LIN {X 0,Y 340.496,Z 607.338,A -85,B 0,C 180,E1 -14141.61,E2 -14141.61} C_VEL
LIN {X 0,Y 341.817,Z 599.412,A -85,B 0,C 180,E1 -14143.677,E2 -14143.677} C_VEL
LIN {X 0,Y 343.018,Z 591.082,A -85,B 0,C 180,E1 -14145.447,E2 -14145.447} C_VEL
LIN {X 0,Y 344.894,Z 580.855,A -85,B 0,C 180,E1 -14147.186,E2 -14147.186} C_VEL
LIN {X 0,Y 346.926,Z 569.542,A -85,B 0,C 180,E1 -14148.759,E2 -14148.759} C_VEL
LIN {X 0,Y 348.186,Z 560.989,A -85,B 0,C 180,E1 -14149.761,E2 -14149.761} C_VEL
LIN {X 0,Y 348.394,Z 548.85,A -85,B 0,C 180,E1 -14151.085,E2 -14151.085} C_VEL
LIN {X 0,Y 347.208,Z 537.307,A -85,B 0,C 180,E1 -14152.297,E2 -14152.297} C_VEL
LIN {X 0,Y 344.797,Z 525.984,A -85,B 0,C 180,E1 -14153.475,E2 -14153.475} C_VEL
LIN {X 0,Y 341.926,Z 516.235,A -85,B 0,C 180,E1 -14154.518,E2 -14154.518} C_VEL
LIN {X 0,Y 340.89,Z 512.472,A -85,B 0,C 180,E1 -14154.888,E2 -14154.888} C_VEL
LIN {X 0,Y 341.816,Z 505.786,A -85,B 0,C 180,E1 -14158.893,E2 -14158.893} C_VEL
LIN {X 0,Y 342.723,Z 500.774,A -85,B 0,C 180,E1 -14162.22,E2 -14162.22} C_VEL
LIN {X 0,Y 343.565,Z 496.904,A -85,B 0,C 180,E1 -14165.09,E2 -14165.09} C_VEL
LIN {X 0,Y 343.924,Z 493.78,A -85,B 0,C 180,E1 -14167.81,E2 -14167.81} C_VEL
LIN {X 0,Y 343.664,Z 490.982,A -85,B 0,C 180,E1 -14170.875,E2 -14170.875} C_VEL
LIN {X 0,Y 343.334,Z 488.645,A -85,B 0,C 180,E1 -14174.238,E2 -14174.238} C_VEL
LIN {X 0,Y 343.008,Z 487.085,A -85,B 0,C 180,E1 -14177.529,E2 -14177.529} C_VEL
LIN {X 0,Y 342.738,Z 486.117,A -85,B 0,C 180,E1 -14181.188,E2 -14181.188} C_VEL
LIN {X 0,Y 342.591,Z 485.893,A -85,B 0,C 180,E1 -14183.494,E2 -14183.494} C_VEL
LIN {X 0,Y 342.084,Z 486.185,A -85,B 0,C 180,E1 -14187.387,E2 -14187.387} C_VEL
LIN {X 0,Y 341.651,Z 486.869,A -85,B 0,C 180,E1 -14190.416,E2 -14190.416} C_VEL
LIN {X 0,Y 341.105,Z 488.27,A -85,B 0,C 180,E1 -14194.363,E2 -14194.363} C_VEL
LIN {X 0,Y 341.043,Z 488.663,A -85,B 0,C 180,E1 -14195.293,E2 -14195.293} C_VEL
LIN {X 0,Y 341.67,Z 490.745,A -85,B 0,C 180,E1 -14195.532,E2 -14195.532} C_VEL
LIN {X 0,Y 344.946,Z 496.905,A -85,B 0,C 180,E1 -14196.469,E2 -14196.469} C_VEL
LIN {X 0,Y 349.037,Z 506.791,A -85,B 0,C 180,E1 -14197.855,E2 -14197.855} C_VEL
LIN {X 0,Y 351.652,Z 516.211,A -85,B 0,C 180,E1 -14199.095,E2 -14199.095} C_VEL
LIN {X 0,Y 352.15,Z 518.968,A -85,B 0,C 180,E1 -14199.449,E2 -14199.449} C_VEL
LIN {X 0,Y 350.175,Z 531.633,A -85,B 0,C 180,E1 -14200.78,E2 -14200.78} C_VEL
LIN {X 0,Y 348.44,Z 541.84,A -85,B 0,C 180,E1 -14202.119,E2 -14202.119} C_VEL
LIN {X 0,Y 346.392,Z 552.222,A -85,B 0,C 180,E1 -14203.801,E2 -14203.801} C_VEL
LIN {X 0,Y 344.984,Z 559.521,A -85,B 0,C 180,E1 -14205.247,E2 -14205.247} C_VEL
LIN {X 0,Y 343.488,Z 566.818,A -85,B 0,C 180,E1 -14206.993,E2 -14206.993} C_VEL
LIN {X 0,Y 342.385,Z 572.658,A -85,B 0,C 180,E1 -14208.755,E2 -14208.755} C_VEL
LIN {X 0,Y 341.397,Z 577.333,A -85,B 0,C 180,E1 -14210.521,E2 -14210.521} C_VEL
LIN {X 0,Y 340.811,Z 580.1,A -85,B 0,C 180,E1 -14211.823,E2 -14211.823} C_VEL
LIN {X 0,Y 340.324,Z 581.969,A -85,B 0,C 180,E1 -14212.883,E2 -14212.883} C_VEL
LIN {X 0,Y 340.031,Z 583.601,A -85,B 0,C 180,E1 -14214.069,E2 -14214.069} C_VEL
LIN {X 0,Y 339.966,Z 584.783,A -85,B 0,C 180,E1 -14215.257,E2 -14215.257} C_VEL
LIN {X 0,Y 339.738,Z 585.596,A -85,B 0,C 180,E1 -14216.442,E2 -14216.442} C_VEL
LIN {X 0,Y 339.542,Z 586.02,A -85,B 0,C 180,E1 -14217.628,E2 -14217.628} C_VEL
LIN {X 0,Y 339.404,Z 586.008,A -85,B 0,C 180,E1 -14218.814,E2 -14218.814} C_VEL
LIN {X 0,Y 339.34,Z 585.584,A -85,B 0,C 180,E1 -14220,E2 -14220} C_VEL
LIN {X 0,Y 339.328,Z 584.764,A -85,B 0,C 180,E1 -14221.187,E2 -14221.187} C_VEL
LIN {X 0,Y 339.33,Z 583.537,A -85,B 0,C 180,E1 -14222.374,E2 -14222.374} C_VEL
LIN {X 0,Y 339.395,Z 580.863,A -85,B 0,C 180,E1 -14224.157,E2 -14224.157} C_VEL
LIN {X 0,Y 339.641,Z 576.209,A -85,B 0,C 180,E1 -14226.32,E2 -14226.32} C_VEL
LIN {X 0,Y 340.017,Z 570.447,A -85,B 0,C 180,E1 -14228.319,E2 -14228.319} C_VEL
LIN {X 0,Y 340.568,Z 563.931,A -85,B 0,C 180,E1 -14230.103,E2 -14230.103} C_VEL
LIN {X 0,Y 341.218,Z 555.819,A -85,B 0,C 180,E1 -14231.887,E2 -14231.887} C_VEL
LIN {X 0,Y 342.13,Z 545.839,A -85,B 0,C 180,E1 -14233.665,E2 -14233.665} C_VEL
LIN {X 0,Y 343.114,Z 535.532,A -85,B 0,C 180,E1 -14235.139,E2 -14235.139} C_VEL
LIN {X 0,Y 343.987,Z 523.853,A -85,B 0,C 180,E1 -14236.498,E2 -14236.498} C_VEL
LIN {X 0,Y 344.746,Z 513.136,A -85,B 0,C 180,E1 -14237.5,E2 -14237.5} C_VEL
LIN {X 0,Y 345.031,Z 508.34,A -85,B 0,C 180,E1 -14237.884,E2 -14237.884} C_VEL
LIN {X 0,Y 342.241,Z 494.577,A -85,B 0,C 180,E1 -14238.919,E2 -14238.919} C_VEL
LIN {X 0,Y 339.504,Z 481.107,A -85,B 0,C 180,E1 -14239.697,E2 -14239.697} C_VEL
LIN {X 0,Y 339.529,Z 477.775,A -85,B 0,C 180,E1 -14243.16,E2 -14243.16} C_VEL
LIN {X 0,Y 339.735,Z 474.171,A -85,B 0,C 180,E1 -14247.072,E2 -14247.072} C_VEL
LIN {X 0,Y 340.04,Z 474.128,A -85,B 0,C 180,E1 -14249.765,E2 -14249.765} C_VEL
LIN {X 0,Y 340.297,Z 474.098,A -85,B 0,C 180,E1 -14252.478,E2 -14252.478} C_VEL
LIN {X 0,Y 340.557,Z 474.061,A -85,B 0,C 180,E1 -14255.299,E2 -14255.299} C_VEL
LIN {X 0,Y 340.706,Z 474.047,A -85,B 0,C 180,E1 -14258.385,E2 -14258.385} C_VEL
LIN {X 0,Y 340.703,Z 474.046,A -85,B 0,C 180,E1 -14262.046,E2 -14262.046} C_VEL
LIN {X 0,Y 340.656,Z 474.054,A -85,B 0,C 180,E1 -14266.227,E2 -14266.227} C_VEL
LIN {X 0,Y 340.692,Z 474.046,A -85,B 0,C 180,E1 -14269.753,E2 -14269.753} C_VEL
LIN {X 0,Y 340.711,Z 474.041,A -85,B 0,C 180,E1 -14273.259,E2 -14273.259} C_VEL
LIN {X 0,Y 340.698,Z 474.049,A -85,B 0,C 180,E1 -14276.154,E2 -14276.154} C_VEL
LIN {X 0,Y 340.779,Z 474.038,A -85,B 0,C 180,E1 -14280.333,E2 -14280.333} C_VEL
LIN {X 0,Y 340.809,Z 474.03,A -85,B 0,C 180,E1 -14283.02,E2 -14283.02} C_VEL
LIN {X 0,Y 340.733,Z 474.039,A -85,B 0,C 180,E1 -14286.927,E2 -14286.927} C_VEL
LIN {X 0,Y 340.799,Z 474.032,A -85,B 0,C 180,E1 -14290.734,E2 -14290.734} C_VEL
LIN {X 0,Y 340.791,Z 474.032,A -85,B 0,C 180,E1 -14293.219,E2 -14293.219} C_VEL
LIN {X 0,Y 340.849,Z 474.025,A -85,B 0,C 180,E1 -14296.891,E2 -14296.891} C_VEL
LIN {X 0,Y 340.933,Z 474.016,A -85,B 0,C 180,E1 -14300.508,E2 -14300.508} C_VEL
LIN {X 0,Y 341.081,Z 473.996,A -85,B 0,C 180,E1 -14302.898,E2 -14302.898} C_VEL
LIN {X 0,Y 341.173,Z 473.987,A -85,B 0,C 180,E1 -14307.639,E2 -14307.639} C_VEL
LIN {X 0,Y 341.3,Z 473.974,A -85,B 0,C 180,E1 -14310,E2 -14310} C_VEL
LIN {X 0,Y 341.173,Z 473.986,A -85,B 0,C 180,E1 -14312.361,E2 -14312.361} C_VEL
LIN {X 0,Y 341.021,Z 474.003,A -85,B 0,C 180,E1 -14317.103,E2 -14317.103} C_VEL
LIN {X 0,Y 340.875,Z 474.022,A -85,B 0,C 180,E1 -14320.694,E2 -14320.694} C_VEL
LIN {X 0,Y 340.868,Z 474.024,A -85,B 0,C 180,E1 -14324.325,E2 -14324.325} C_VEL
LIN {X 0,Y 340.843,Z 474.027,A -85,B 0,C 180,E1 -14328.467,E2 -14328.467} C_VEL
LIN {X 0,Y 340.726,Z 474.045,A -85,B 0,C 180,E1 -14331.843,E2 -14331.843} C_VEL
LIN {X 0,Y 340.776,Z 474.038,A -85,B 0,C 180,E1 -14335.664,E2 -14335.664} C_VEL
LIN {X 0,Y 340.732,Z 474.041,A -85,B 0,C 180,E1 -14338.321,E2 -14338.321} C_VEL
LIN {X 0,Y 340.702,Z 474.043,A -85,B 0,C 180,E1 -14341.044,E2 -14341.044} C_VEL
LIN {X 0,Y 340.723,Z 474.042,A -85,B 0,C 180,E1 -14345.278,E2 -14345.278} C_VEL
LIN {X 0,Y 340.716,Z 474.042,A -85,B 0,C 180,E1 -14348.386,E2 -14348.386} C_VEL
LIN {X 0,Y 340.703,Z 474.046,A -85,B 0,C 180,E1 -14352.045,E2 -14352.045} C_VEL
LIN {X 0,Y 340.656,Z 474.05,A -85,B 0,C 180,E1 -14356.227,E2 -14356.227} C_VEL
LIN {X 0,Y 340.693,Z 474.05,A -85,B 0,C 180,E1 -14359.752,E2 -14359.752} C_VEL
LIN {X 0,Y 340.687,Z 474.046,A -85,B 0,C 180,E1 -14363.256,E2 -14363.256} C_VEL
LIN {X 0,Y 340.533,Z 474.066,A -85,B 0,C 180,E1 -14366.135,E2 -14366.135} C_VEL
LIN {X 0,Y 340.22,Z 474.103,A -85,B 0,C 180,E1 -14368.906,E2 -14368.906} C_VEL
LIN {X 0,Y 339.997,Z 474.131,A -85,B 0,C 180,E1 -14370.677,E2 -14370.677} C_VEL
LIN {X 0,Y 339.191,Z 474.237,A -85,B 0,C 180,E1 -14371.664,E2 -14371.664} C_VEL
LIN {X 0,Y 336.119,Z 474.617,A -85,B 0,C 180,E1 -14373.265,E2 -14373.265} C_VEL
LIN {X 0,Y 333.569,Z 475.163,A -85,B 0,C 180,E1 -14374.556,E2 -14374.556} C_VEL
LIN {X 0,Y 332.468,Z 475.886,A -85,B 0,C 180,E1 -14375.552,E2 -14375.552} C_VEL
LIN {X 0,Y 332.372,Z 476.217,A -85,B 0,C 180,E1 -14375.888,E2 -14375.888} C_VEL
LIN {X 0,Y 332.378,Z 480.517,A -85,B 0,C 180,E1 -14379.903,E2 -14379.903} C_VEL
LIN {X 0,Y 332.379,Z 480.826,A -85,B 0,C 180,E1 -14380.185,E2 -14380.185} C_VEL
LIN {X 0,Y 335.524,Z 496.725,A -85,B 0,C 180,E1 -14381.146,E2 -14381.146} C_VEL
LIN {X 0,Y 337.973,Z 509.393,A -85,B 0,C 180,E1 -14382.138,E2 -14382.138} C_VEL
LIN {X 0,Y 337.084,Z 521.968,A -85,B 0,C 180,E1 -14383.274,E2 -14383.274} C_VEL
LIN {X 0,Y 336.139,Z 534.349,A -85,B 0,C 180,E1 -14384.694,E2 -14384.694} C_VEL
LIN {X 0,Y 335.24,Z 543.893,A -85,B 0,C 180,E1 -14386.049,E2 -14386.049} C_VEL
LIN {X 0,Y 334.219,Z 554.344,A -85,B 0,C 180,E1 -14387.861,E2 -14387.861} C_VEL
LIN {X 0,Y 333.528,Z 562.727,A -85,B 0,C 180,E1 -14389.682,E2 -14389.682} C_VEL
LIN {X 0,Y 332.939,Z 569.529,A -85,B 0,C 180,E1 -14391.502,E2 -14391.502} C_VEL
LIN {X 0,Y 332.624,Z 574.779,A -85,B 0,C 180,E1 -14393.249,E2 -14393.249} C_VEL
LIN {X 0,Y 332.393,Z 579.258,A -85,B 0,C 180,E1 -14395.148,E2 -14395.148} C_VEL
LIN {X 0,Y 332.264,Z 581.475,A -85,B 0,C 180,E1 -14396.362,E2 -14396.362} C_VEL
LIN {X 0,Y 332.225,Z 583.247,A -85,B 0,C 180,E1 -14397.575,E2 -14397.575} C_VEL
LIN {X 0,Y 332.196,Z 584.613,A -85,B 0,C 180,E1 -14398.787,E2 -14398.787} C_VEL
LIN {X 0,Y 332.235,Z 585.528,A -85,B 0,C 180,E1 -14400,E2 -14400} C_VEL
LIN {X 0,Y 332.48,Z 586.136,A -85,B 0,C 180,E1 -14402.423,E2 -14402.423} C_VEL
LIN {X 0,Y 332.69,Z 585.836,A -85,B 0,C 180,E1 -14403.633,E2 -14403.633} C_VEL
LIN {X 0,Y 332.841,Z 585.101,A -85,B 0,C 180,E1 -14404.845,E2 -14404.845} C_VEL
LIN {X 0,Y 332.912,Z 583.989,A -85,B 0,C 180,E1 -14406.059,E2 -14406.059} C_VEL
LIN {X 0,Y 333.748,Z 580.936,A -85,B 0,C 180,E1 -14408.222,E2 -14408.222} C_VEL
LIN {X 0,Y 334.66,Z 576.679,A -85,B 0,C 180,E1 -14410.282,E2 -14410.282} C_VEL
LIN {X 0,Y 335.8,Z 571.755,A -85,B 0,C 180,E1 -14412.081,E2 -14412.081} C_VEL
LIN {X 0,Y 337.049,Z 565.63,A -85,B 0,C 180,E1 -14413.874,E2 -14413.874} C_VEL
LIN {X 0,Y 338.647,Z 558.164,A -85,B 0,C 180,E1 -14415.652,E2 -14415.652} C_VEL
LIN {X 0,Y 340.629,Z 548.877,A -85,B 0,C 180,E1 -14417.408,E2 -14417.408} C_VEL
LIN {X 0,Y 342.603,Z 538.877,A -85,B 0,C 180,E1 -14418.944,E2 -14418.944} C_VEL
LIN {X 0,Y 344.492,Z 528.159,A -85,B 0,C 180,E1 -14420.293,E2 -14420.293} C_VEL
LIN {X 0,Y 345.869,Z 519.994,A -85,B 0,C 180,E1 -14421.142,E2 -14421.142} C_VEL
LIN {X 0,Y 344.09,Z 511.553,A -85,B 0,C 180,E1 -14422.28,E2 -14422.28} C_VEL
LIN {X 0,Y 340.643,Z 501.465,A -85,B 0,C 180,E1 -14423.708,E2 -14423.708} C_VEL
LIN {X 0,Y 335.961,Z 491.247,A -85,B 0,C 180,E1 -14425.26,E2 -14425.26} C_VEL
LIN {X 0,Y 334.34,Z 488.16,A -85,B 0,C 180,E1 -14425.755,E2 -14425.755} C_VEL
LIN {X 0,Y 334.158,Z 487.37,A -85,B 0,C 180,E1 -14425.866,E2 -14425.866} C_VEL
LIN {X 0,Y 334.333,Z 484.941,A -85,B 0,C 180,E1 -14428.913,E2 -14428.913} C_VEL
LIN {X 0,Y 334.598,Z 482.863,A -85,B 0,C 180,E1 -14431.675,E2 -14431.675} C_VEL
LIN {X 0,Y 334.724,Z 480.616,A -85,B 0,C 180,E1 -14435.029,E2 -14435.029} C_VEL
LIN {X 0,Y 334.588,Z 479.264,A -85,B 0,C 180,E1 -14437.528,E2 -14437.528} C_VEL
LIN {X 0,Y 334.37,Z 477.929,A -85,B 0,C 180,E1 -14440.828,E2 -14440.828} C_VEL
LIN {X 0,Y 334.191,Z 477.226,A -85,B 0,C 180,E1 -14444.355,E2 -14444.355} C_VEL
LIN {X 0,Y 334.119,Z 477.409,A -85,B 0,C 180,E1 -14446.387,E2 -14446.387} C_VEL
LIN {X 0,Y 335.222,Z 483.366,A -85,B 0,C 180,E1 -14450.197,E2 -14450.197} C_VEL
LIN {X 0,Y 335.855,Z 487.414,A -85,B 0,C 180,E1 -14452.672,E2 -14452.672} C_VEL
LIN {X 0,Y 335.789,Z 490.904,A -85,B 0,C 180,E1 -14454.712,E2 -14454.712} C_VEL
LIN {X 0,Y 334.967,Z 497.396,A -85,B 0,C 180,E1 -14458.363,E2 -14458.363} C_VEL
LIN {X 0,Y 334.076,Z 504.808,A -85,B 0,C 180,E1 -14462.431,E2 -14462.431} C_VEL
LIN {X 0,Y 333.699,Z 508.242,A -85,B 0,C 180,E1 -14464.212,E2 -14464.212} C_VEL
LIN {X 0,Y 334.485,Z 512.006,A -85,B 0,C 180,E1 -14464.578,E2 -14464.578} C_VEL
LIN {X 0,Y 335.342,Z 514.335,A -85,B 0,C 180,E1 -14464.855,E2 -14464.855} C_VEL
LIN {X 0,Y 338.443,Z 526.565,A -85,B 0,C 180,E1 -14466.171,E2 -14466.171} C_VEL
LIN {X 0,Y 340.605,Z 539.432,A -85,B 0,C 180,E1 -14467.544,E2 -14467.544} C_VEL
LIN {X 0,Y 341.392,Z 550.711,A -85,B 0,C 180,E1 -14468.783,E2 -14468.783} C_VEL
LIN {X 0,Y 341.006,Z 563.3,A -85,B 0,C 180,E1 -14470.276,E2 -14470.276} C_VEL
LIN {X 0,Y 339.006,Z 574.502,A -85,B 0,C 180,E1 -14471.726,E2 -14471.726} C_VEL
LIN {X 0,Y 337.173,Z 584.837,A -85,B 0,C 180,E1 -14473.374,E2 -14473.374} C_VEL
LIN {X 0,Y 335.767,Z 592.423,A -85,B 0,C 180,E1 -14474.833,E2 -14474.833} C_VEL
LIN {X 0,Y 334.486,Z 600.221,A -85,B 0,C 180,E1 -14476.637,E2 -14476.637} C_VEL
LIN {X 0,Y 333.373,Z 606.607,A -85,B 0,C 180,E1 -14478.447,E2 -14478.447} C_VEL
LIN {X 0,Y 332.716,Z 611.78,A -85,B 0,C 180,E1 -14480.271,E2 -14480.271} C_VEL
LIN {X 0,Y 332.326,Z 615.858,A -85,B 0,C 180,E1 -14482.099,E2 -14482.099} C_VEL
LIN {X 0,Y 332.18,Z 618.907,A -85,B 0,C 180,E1 -14483.928,E2 -14483.928} C_VEL
LIN {X 0,Y 332.114,Z 620.392,A -85,B 0,C 180,E1 -14485.144,E2 -14485.144} C_VEL
LIN {X 0,Y 332.104,Z 621.472,A -85,B 0,C 180,E1 -14486.36,E2 -14486.36} C_VEL
LIN {X 0,Y 332.293,Z 623.081,A -85,B 0,C 180,E1 -14488.788,E2 -14488.788} C_VEL
LIN {X 0,Y 332.277,Z 623.714,A -85,B 0,C 180,E1 -14490,E2 -14490} C_VEL
LIN {X 0,Y 332.252,Z 623.93,A -85,B 0,C 180,E1 -14491.212,E2 -14491.212} C_VEL
LIN {X 0,Y 332.081,Z 623.725,A -85,B 0,C 180,E1 -14492.426,E2 -14492.426} C_VEL
LIN {X 0,Y 332.058,Z 623.108,A -85,B 0,C 180,E1 -14493.64,E2 -14493.64} C_VEL
LIN {X 0,Y 332.045,Z 620.869,A -85,B 0,C 180,E1 -14495.848,E2 -14495.848} C_VEL
LIN {X 0,Y 332.321,Z 617.551,A -85,B 0,C 180,E1 -14497.901,E2 -14497.901} C_VEL
LIN {X 0,Y 332.748,Z 613.523,A -85,B 0,C 180,E1 -14499.728,E2 -14499.728} C_VEL
LIN {X 0,Y 333.403,Z 608.444,A -85,B 0,C 180,E1 -14501.552,E2 -14501.552} C_VEL
LIN {X 0,Y 334.727,Z 601.005,A -85,B 0,C 180,E1 -14503.663,E2 -14503.663} C_VEL
LIN {X 0,Y 335.98,Z 593.086,A -85,B 0,C 180,E1 -14505.468,E2 -14505.468} C_VEL
LIN {X 0,Y 337.879,Z 583.553,A -85,B 0,C 180,E1 -14507.242,E2 -14507.242} C_VEL
LIN {X 0,Y 339.924,Z 572.979,A -85,B 0,C 180,E1 -14508.848,E2 -14508.848} C_VEL
LIN {X 0,Y 341.693,Z 562.538,A -85,B 0,C 180,E1 -14510.152,E2 -14510.152} C_VEL
LIN {X 0,Y 342.125,Z 551.121,A -85,B 0,C 180,E1 -14511.491,E2 -14511.491} C_VEL
LIN {X 0,Y 341.157,Z 539.755,A -85,B 0,C 180,E1 -14512.757,E2 -14512.757} C_VEL
LIN {X 0,Y 339.073,Z 528.891,A -85,B 0,C 180,E1 -14513.987,E2 -14513.987} C_VEL
LIN {X 0,Y 335.758,Z 516.942,A -85,B 0,C 180,E1 -14515.361,E2 -14515.361} C_VEL
LIN {X 0,Y 334.191,Z 512.494,A -85,B 0,C 180,E1 -14515.897,E2 -14515.897} C_VEL
LIN {X 0,Y 334.081,Z 511.612,A -85,B 0,C 180,E1 -14516.01,E2 -14516.01} C_VEL
LIN {X 0,Y 334.958,Z 505.999,A -85,B 0,C 180,E1 -14519.543,E2 -14519.543} C_VEL
LIN {X 0,Y 336.044,Z 500.735,A -85,B 0,C 180,E1 -14523.222,E2 -14523.222} C_VEL
LIN {X 0,Y 336.707,Z 497.527,A -85,B 0,C 180,E1 -14525.763,E2 -14525.763} C_VEL
LIN {X 0,Y 336.986,Z 495.505,A -85,B 0,C 180,E1 -14527.579,E2 -14527.579} C_VEL
LIN {X 0,Y 336.771,Z 492.993,A -85,B 0,C 180,E1 -14530.311,E2 -14530.311} C_VEL
LIN {X 0,Y 336.456,Z 490.624,A -85,B 0,C 180,E1 -14533.576,E2 -14533.576} C_VEL
LIN {X 0,Y 336.131,Z 488.849,A -85,B 0,C 180,E1 -14537.038,E2 -14537.038} C_VEL
LIN {X 0,Y 335.843,Z 487.754,A -85,B 0,C 180,E1 -14540.74,E2 -14540.74} C_VEL
LIN {X 0,Y 335.563,Z 487.416,A -85,B 0,C 180,E1 -14544.096,E2 -14544.096} C_VEL
LIN {X 0,Y 335.191,Z 487.593,A -85,B 0,C 180,E1 -14547.002,E2 -14547.002} C_VEL
LIN {X 0,Y 334.819,Z 488.108,A -85,B 0,C 180,E1 -14549.75,E2 -14549.75} C_VEL
LIN {X 0,Y 334.374,Z 488.911,A -85,B 0,C 180,E1 -14552.458,E2 -14552.458} C_VEL
LIN {X 0,Y 334.19,Z 489.753,A -85,B 0,C 180,E1 -14554.235,E2 -14554.235} C_VEL
LIN {X 0,Y 334.84,Z 491.695,A -85,B 0,C 180,E1 -14554.493,E2 -14554.493} C_VEL
LIN {X 0,Y 336.559,Z 494.566,A -85,B 0,C 180,E1 -14555,E2 -14555} C_VEL
LIN {X 0,Y 341.643,Z 505.533,A -85,B 0,C 180,E1 -14556.726,E2 -14556.726} C_VEL
LIN {X 0,Y 344.431,Z 513.763,A -85,B 0,C 180,E1 -14557.939,E2 -14557.939} C_VEL
LIN {X 0,Y 345.962,Z 520.424,A -85,B 0,C 180,E1 -14558.865,E2 -14558.865} C_VEL
LIN {X 0,Y 344.002,Z 532.862,A -85,B 0,C 180,E1 -14560.242,E2 -14560.242} C_VEL
LIN {X 0,Y 341.96,Z 543.699,A -85,B 0,C 180,E1 -14561.735,E2 -14561.735} C_VEL
LIN {X 0,Y 339.778,Z 554.044,A -85,B 0,C 180,E1 -14563.477,E2 -14563.477} C_VEL
LIN {X 0,Y 337.997,Z 562.331,A -85,B 0,C 180,E1 -14565.243,E2 -14565.243} C_VEL
LIN {X 0,Y 336.297,Z 570.142,A -85,B 0,C 180,E1 -14567.325,E2 -14567.325} C_VEL
LIN {X 0,Y 335.006,Z 575.464,A -85,B 0,C 180,E1 -14569.117,E2 -14569.117} C_VEL
LIN {X 0,Y 334.179,Z 579.617,A -85,B 0,C 180,E1 -14570.925,E2 -14570.925} C_VEL
LIN {X 0,Y 333.327,Z 582.773,A -85,B 0,C 180,E1 -14572.732,E2 -14572.732} C_VEL
LIN {X 0,Y 332.997,Z 584.305,A -85,B 0,C 180,E1 -14573.943,E2 -14573.943} C_VEL
LIN {X 0,Y 332.933,Z 585.431,A -85,B 0,C 180,E1 -14575.157,E2 -14575.157} C_VEL
LIN {X 0,Y 332.699,Z 586.188,A -85,B 0,C 180,E1 -14576.367,E2 -14576.367} C_VEL
LIN {X 0,Y 332.491,Z 586.523,A -85,B 0,C 180,E1 -14577.577,E2 -14577.577} C_VEL
LIN {X 0,Y 332.346,Z 586.435,A -85,B 0,C 180,E1 -14578.789,E2 -14578.789} C_VEL
LIN {X 0,Y 332.261,Z 585.954,A -85,B 0,C 180,E1 -14580,E2 -14580} C_VEL
LIN {X 0,Y 332.236,Z 585.078,A -85,B 0,C 180,E1 -14581.212,E2 -14581.212} C_VEL
LIN {X 0,Y 332.235,Z 583.755,A -85,B 0,C 180,E1 -14582.425,E2 -14582.425} C_VEL
LIN {X 0,Y 332.329,Z 580.982,A -85,B 0,C 180,E1 -14584.245,E2 -14584.245} C_VEL
LIN {X 0,Y 332.528,Z 577.163,A -85,B 0,C 180,E1 -14586.066,E2 -14586.066} C_VEL
LIN {X 0,Y 332.844,Z 572.204,A -85,B 0,C 180,E1 -14587.889,E2 -14587.889} C_VEL
LIN {X 0,Y 333.429,Z 564.814,A -85,B 0,C 180,E1 -14590.015,E2 -14590.015} C_VEL
LIN {X 0,Y 334.106,Z 556.824,A -85,B 0,C 180,E1 -14591.835,E2 -14591.835} C_VEL
LIN {X 0,Y 335.012,Z 546.946,A -85,B 0,C 180,E1 -14593.651,E2 -14593.651} C_VEL
LIN {X 0,Y 335.997,Z 536.831,A -85,B 0,C 180,E1 -14595.157,E2 -14595.157} C_VEL
LIN {X 0,Y 336.898,Z 525.046,A -85,B 0,C 180,E1 -14596.579,E2 -14596.579} C_VEL
LIN {X 0,Y 337.777,Z 513.253,A -85,B 0,C 180,E1 -14597.716,E2 -14597.716} C_VEL
LIN {X 0,Y 337.941,Z 508.65,A -85,B 0,C 180,E1 -14598.099,E2 -14598.099} C_VEL
LIN {X 0,Y 335.191,Z 495.352,A -85,B 0,C 180,E1 -14599.12,E2 -14599.12} C_VEL
LIN {X 0,Y 332.429,Z 481.496,A -85,B 0,C 180,E1 -14599.932,E2 -14599.932} C_VEL
LIN {X 0,Y 332.467,Z 477.936,A -85,B 0,C 180,E1 -14603.681,E2 -14603.681} C_VEL
LIN {X 0,Y 332.597,Z 475.452,A -85,B 0,C 180,E1 -14606.344,E2 -14606.344} C_VEL
LIN {X 0,Y 332.736,Z 475.044,A -85,B 0,C 180,E1 -14607.69,E2 -14607.69} C_VEL
LIN {X 0,Y 333.033,Z 475.003,A -85,B 0,C 180,E1 -14610.43,E2 -14610.43} C_VEL
LIN {X 0,Y 333.306,Z 474.964,A -85,B 0,C 180,E1 -14613.246,E2 -14613.246} C_VEL
LIN {X 0,Y 333.635,Z 474.924,A -85,B 0,C 180,E1 -14616.825,E2 -14616.825} C_VEL
LIN {X 0,Y 333.651,Z 474.923,A -85,B 0,C 180,E1 -14620.685,E2 -14620.685} C_VEL
LIN {X 0,Y 333.598,Z 474.933,A -85,B 0,C 180,E1 -14624.251,E2 -14624.251} C_VEL
LIN {X 0,Y 333.645,Z 474.923,A -85,B 0,C 180,E1 -14627.619,E2 -14627.619} C_VEL
LIN {X 0,Y 333.658,Z 474.92,A -85,B 0,C 180,E1 -14631.202,E2 -14631.202} C_VEL
LIN {X 0,Y 333.681,Z 474.92,A -85,B 0,C 180,E1 -14633.861,E2 -14633.861} C_VEL
LIN {X 0,Y 333.65,Z 474.921,A -85,B 0,C 180,E1 -14637.413,E2 -14637.413} C_VEL
LIN {X 0,Y 333.715,Z 474.913,A -85,B 0,C 180,E1 -14641.028,E2 -14641.028} C_VEL
LIN {X 0,Y 333.74,Z 474.912,A -85,B 0,C 180,E1 -14643.754,E2 -14643.754} C_VEL
LIN {X 0,Y 333.724,Z 474.916,A -85,B 0,C 180,E1 -14647.914,E2 -14647.914} C_VEL
LIN {X 0,Y 333.799,Z 474.904,A -85,B 0,C 180,E1 -14651.59,E2 -14651.59} C_VEL
LIN {X 0,Y 333.813,Z 474.902,A -85,B 0,C 180,E1 -14655.577,E2 -14655.577} C_VEL
LIN {X 0,Y 333.839,Z 474.897,A -85,B 0,C 180,E1 -14659.078,E2 -14659.078} C_VEL
LIN {X 0,Y 334.031,Z 474.874,A -85,B 0,C 180,E1 -14662.748,E2 -14662.748} C_VEL
LIN {X 0,Y 333.815,Z 474.901,A -85,B 0,C 180,E1 -14665.169,E2 -14665.169} C_VEL
LIN {X 0,Y 334.11,Z 474.866,A -85,B 0,C 180,E1 -14667.589,E2 -14667.589} C_VEL
LIN {X 0,Y 334.251,Z 474.852,A -85,B 0,C 180,E1 -14670,E2 -14670} C_VEL
LIN {X 0,Y 334.11,Z 474.866,A -85,B 0,C 180,E1 -14672.411,E2 -14672.411} C_VEL
LIN {X 0,Y 334.004,Z 474.882,A -85,B 0,C 180,E1 -14676.039,E2 -14676.039} C_VEL
LIN {X 0,Y 333.853,Z 474.899,A -85,B 0,C 180,E1 -14679.695,E2 -14679.695} C_VEL
LIN {X 0,Y 333.802,Z 474.903,A -85,B 0,C 180,E1 -14683.391,E2 -14683.391} C_VEL
LIN {X 0,Y 333.751,Z 474.909,A -85,B 0,C 180,E1 -14687.146,E2 -14687.146} C_VEL
LIN {X 0,Y 333.74,Z 474.914,A -85,B 0,C 180,E1 -14689.69,E2 -14689.69} C_VEL
LIN {X 0,Y 333.676,Z 474.921,A -85,B 0,C 180,E1 -14693.59,E2 -14693.59} C_VEL
LIN {X 0,Y 333.739,Z 474.912,A -85,B 0,C 180,E1 -14696.246,E2 -14696.246} C_VEL
LIN {X 0,Y 333.694,Z 474.916,A -85,B 0,C 180,E1 -14698.974,E2 -14698.974} C_VEL
LIN {X 0,Y 333.65,Z 474.921,A -85,B 0,C 180,E1 -14702.587,E2 -14702.587} C_VEL
LIN {X 0,Y 333.681,Z 474.92,A -85,B 0,C 180,E1 -14706.138,E2 -14706.138} C_VEL
LIN {X 0,Y 333.651,Z 474.922,A -85,B 0,C 180,E1 -14709.192,E2 -14709.192} C_VEL
LIN {X 0,Y 333.636,Z 474.923,A -85,B 0,C 180,E1 -14712.5,E2 -14712.5} C_VEL
LIN {X 0,Y 333.601,Z 474.931,A -85,B 0,C 180,E1 -14715.955,E2 -14715.955} C_VEL
LIN {X 0,Y 333.651,Z 474.923,A -85,B 0,C 180,E1 -14719.315,E2 -14719.315} C_VEL
LIN {X 0,Y 333.65,Z 474.922,A -85,B 0,C 180,E1 -14723.172,E2 -14723.172} C_VEL
LIN {X 0,Y 333.424,Z 474.949,A -85,B 0,C 180,E1 -14726.767,E2 -14726.767} C_VEL
LIN {X 0,Y 332.955,Z 475.008,A -85,B 0,C 180,E1 -14730.656,E2 -14730.656} C_VEL
LIN {X 0,Y 332.487,Z 475.069,A -85,B 0,C 180,E1 -14734.321,E2 -14734.321} C_VEL
LIN {X 0,Y 332.426,Z 475.264,A -85,B 0,C 180,E1 -14734.986,E2 -14734.986} C_VEL
LIN {X 0,Y 332.372,Z 476.217,A -85,B 0,C 180,E1 -14735.888,E2 -14735.888} C_VEL
LIN {X 0,Y 331.679,Z 476.986,A -85,B 0,C 180,E1 -14736.548,E2 -14736.548} C_VEL
LIN {X 0,Y 328.822,Z 478.348,A -85,B 0,C 180,E1 -14737.577,E2 -14737.577} C_VEL
LIN {X 0,Y 325.963,Z 479.714,A -85,B 0,C 180,E1 -14738.623,E2 -14738.623} C_VEL
LIN {X 0,Y 325.292,Z 480.498,A -85,B 0,C 180,E1 -14739.302,E2 -14739.302} C_VEL
LIN {X 0,Y 325.306,Z 481.171,A -85,B 0,C 180,E1 -14739.929,E2 -14739.929} C_VEL
LIN {X 0,Y 328.254,Z 496.354,A -85,B 0,C 180,E1 -14740.862,E2 -14740.862} C_VEL
LIN {X 0,Y 330.77,Z 509.322,A -85,B 0,C 180,E1 -14741.896,E2 -14741.896} C_VEL
LIN {X 0,Y 330.54,Z 516.482,A -85,B 0,C 180,E1 -14742.522,E2 -14742.522} C_VEL
LIN {X 0,Y 329.538,Z 529.554,A -85,B 0,C 180,E1 -14743.904,E2 -14743.904} C_VEL
LIN {X 0,Y 328.582,Z 540.013,A -85,B 0,C 180,E1 -14745.286,E2 -14745.286} C_VEL
LIN {X 0,Y 327.556,Z 550.469,A -85,B 0,C 180,E1 -14746.98,E2 -14746.98} C_VEL
LIN {X 0,Y 326.74,Z 559.698,A -85,B 0,C 180,E1 -14748.838,E2 -14748.838} C_VEL
LIN {X 0,Y 326.088,Z 567.169,A -85,B 0,C 180,E1 -14750.697,E2 -14750.697} C_VEL
LIN {X 0,Y 325.636,Z 573.186,A -85,B 0,C 180,E1 -14752.559,E2 -14752.559} C_VEL
LIN {X 0,Y 325.39,Z 577.947,A -85,B 0,C 180,E1 -14754.422,E2 -14754.422} C_VEL
LIN {X 0,Y 325.19,Z 581.588,A -85,B 0,C 180,E1 -14756.282,E2 -14756.282} C_VEL
LIN {X 0,Y 325.131,Z 583.422,A -85,B 0,C 180,E1 -14757.522,E2 -14757.522} C_VEL
LIN {X 0,Y 325.101,Z 584.85,A -85,B 0,C 180,E1 -14758.761,E2 -14758.761} C_VEL
LIN {X 0,Y 325.144,Z 585.873,A -85,B 0,C 180,E1 -14760,E2 -14760} C_VEL
LIN {X 0,Y 325.238,Z 586.439,A -85,B 0,C 180,E1 -14761.238,E2 -14761.238} C_VEL
LIN {X 0,Y 325.412,Z 586.605,A -85,B 0,C 180,E1 -14762.475,E2 -14762.475} C_VEL
LIN {X 0,Y 325.63,Z 586.378,A -85,B 0,C 180,E1 -14763.712,E2 -14763.712} C_VEL
LIN {X 0,Y 325.793,Z 585.747,A -85,B 0,C 180,E1 -14764.95,E2 -14764.95} C_VEL
LIN {X 0,Y 325.885,Z 584.708,A -85,B 0,C 180,E1 -14766.19,E2 -14766.19} C_VEL
LIN {X 0,Y 326.781,Z 581.813,A -85,B 0,C 180,E1 -14768.383,E2 -14768.383} C_VEL
LIN {X 0,Y 327.748,Z 577.71,A -85,B 0,C 180,E1 -14770.502,E2 -14770.502} C_VEL
LIN {X 0,Y 328.968,Z 572.965,A -85,B 0,C 180,E1 -14772.335,E2 -14772.335} C_VEL
LIN {X 0,Y 330.32,Z 567.053,A -85,B 0,C 180,E1 -14774.163,E2 -14774.163} C_VEL
LIN {X 0,Y 331.997,Z 559.754,A -85,B 0,C 180,E1 -14775.973,E2 -14775.973} C_VEL
LIN {X 0,Y 334.098,Z 550.84,A -85,B 0,C 180,E1 -14777.759,E2 -14777.759} C_VEL
LIN {X 0,Y 336.469,Z 539.837,A -85,B 0,C 180,E1 -14779.524,E2 -14779.524} C_VEL
LIN {X 0,Y 338.565,Z 528.71,A -85,B 0,C 180,E1 -14780.95,E2 -14780.95} C_VEL
LIN {X 0,Y 339.755,Z 521.85,A -85,B 0,C 180,E1 -14781.7,E2 -14781.7} C_VEL
LIN {X 0,Y 338.006,Z 513.498,A -85,B 0,C 180,E1 -14782.916,E2 -14782.916} C_VEL
LIN {X 0,Y 334.622,Z 503.528,A -85,B 0,C 180,E1 -14784.452,E2 -14784.452} C_VEL
LIN {X 0,Y 331.443,Z 496.294,A -85,B 0,C 180,E1 -14785.628,E2 -14785.628} C_VEL
LIN {X 0,Y 329.103,Z 491.959,A -85,B 0,C 180,E1 -14786.418,E2 -14786.418} C_VEL
LIN {X 0,Y 327.493,Z 488.852,A -85,B 0,C 180,E1 -14786.969,E2 -14786.969} C_VEL
LIN {X 0,Y 327.325,Z 488.186,A -85,B 0,C 180,E1 -14787.059,E2 -14787.059} C_VEL
LIN {X 0,Y 327.697,Z 485.292,A -85,B 0,C 180,E1 -14790.979,E2 -14790.979} C_VEL
LIN {X 0,Y 327.89,Z 483.403,A -85,B 0,C 180,E1 -14793.868,E2 -14793.868} C_VEL
LIN {X 0,Y 327.869,Z 481.787,A -85,B 0,C 180,E1 -14796.883,E2 -14796.883} C_VEL
LIN {X 0,Y 327.698,Z 480.572,A -85,B 0,C 180,E1 -14800.046,E2 -14800.046} C_VEL
LIN {X 0,Y 327.575,Z 479.93,A -85,B 0,C 180,E1 -14803.357,E2 -14803.357} C_VEL
LIN {X 0,Y 327.57,Z 479.849,A -85,B 0,C 180,E1 -14805.073,E2 -14805.073} C_VEL
LIN {X 0,Y 327.456,Z 480.329,A -85,B 0,C 180,E1 -14807.585,E2 -14807.585} C_VEL
LIN {X 0,Y 328.261,Z 484.712,A -85,B 0,C 180,E1 -14810.422,E2 -14810.422} C_VEL
LIN {X 0,Y 328.888,Z 489.273,A -85,B 0,C 180,E1 -14813.249,E2 -14813.249} C_VEL
LIN {X 0,Y 328.581,Z 493.046,A -85,B 0,C 180,E1 -14815.472,E2 -14815.472} C_VEL
LIN {X 0,Y 327.677,Z 499.36,A -85,B 0,C 180,E1 -14819.084,E2 -14819.084} C_VEL
LIN {X 0,Y 326.968,Z 505.398,A -85,B 0,C 180,E1 -14822.475,E2 -14822.475} C_VEL
LIN {X 0,Y 326.883,Z 506.414,A -85,B 0,C 180,E1 -14822.922,E2 -14822.922} C_VEL
LIN {X 0,Y 327.604,Z 510.053,A -85,B 0,C 180,E1 -14823.311,E2 -14823.311} C_VEL
LIN {X 0,Y 328.667,Z 512.658,A -85,B 0,C 180,E1 -14823.669,E2 -14823.669} C_VEL
LIN {X 0,Y 332.104,Z 526.167,A -85,B 0,C 180,E1 -14825.25,E2 -14825.25} C_VEL
LIN {X 0,Y 334.288,Z 539.435,A -85,B 0,C 180,E1 -14826.776,E2 -14826.776} C_VEL
LIN {X 0,Y 335.131,Z 550.563,A -85,B 0,C 180,E1 -14828.083,E2 -14828.083} C_VEL
LIN {X 0,Y 334.614,Z 563.818,A -85,B 0,C 180,E1 -14829.723,E2 -14829.723} C_VEL
LIN {X 0,Y 332.566,Z 574.699,A -85,B 0,C 180,E1 -14831.199,E2 -14831.199} C_VEL
LIN {X 0,Y 330.439,Z 585.664,A -85,B 0,C 180,E1 -14833.027,E2 -14833.027} C_VEL
LIN {X 0,Y 328.945,Z 593.029,A -85,B 0,C 180,E1 -14834.51,E2 -14834.51} C_VEL
LIN {X 0,Y 327.355,Z 601.696,A -85,B 0,C 180,E1 -14836.656,E2 -14836.656} C_VEL
LIN {X 0,Y 326.393,Z 606.798,A -85,B 0,C 180,E1 -14838.196,E2 -14838.196} C_VEL
LIN {X 0,Y 325.705,Z 611.826,A -85,B 0,C 180,E1 -14840.06,E2 -14840.06} C_VEL
LIN {X 0,Y 325.255,Z 615.76,A -85,B 0,C 180,E1 -14841.926,E2 -14841.926} C_VEL
LIN {X 0,Y 325.102,Z 618.902,A -85,B 0,C 180,E1 -14843.945,E2 -14843.945} C_VEL
LIN {X 0,Y 325.027,Z 621.129,A -85,B 0,C 180,E1 -14846.281,E2 -14846.281} C_VEL
LIN {X 0,Y 325.234,Z 622.469,A -85,B 0,C 180,E1 -14848.762,E2 -14848.762} C_VEL
LIN {X 0,Y 325.219,Z 623.191,A -85,B 0,C 180,E1 -14850,E2 -14850} C_VEL
LIN {X 0,Y 325.17,Z 623.453,A -85,B 0,C 180,E1 -14851.238,E2 -14851.238} C_VEL
LIN {X 0,Y 324.98,Z 622.741,A -85,B 0,C 180,E1 -14853.72,E2 -14853.72} C_VEL
LIN {X 0,Y 324.962,Z 620.843,A -85,B 0,C 180,E1 -14855.818,E2 -14855.818} C_VEL
LIN {X 0,Y 325.252,Z 617.449,A -85,B 0,C 180,E1 -14858.074,E2 -14858.074} C_VEL
LIN {X 0,Y 325.737,Z 613.566,A -85,B 0,C 180,E1 -14859.939,E2 -14859.939} C_VEL
LIN {X 0,Y 326.42,Z 608.609,A -85,B 0,C 180,E1 -14861.803,E2 -14861.803} C_VEL
LIN {X 0,Y 327.844,Z 601.33,A -85,B 0,C 180,E1 -14863.955,E2 -14863.955} C_VEL
LIN {X 0,Y 329.16,Z 593.754,A -85,B 0,C 180,E1 -14865.788,E2 -14865.788} C_VEL
LIN {X 0,Y 331.169,Z 584.427,A -85,B 0,C 180,E1 -14867.603,E2 -14867.603} C_VEL
LIN {X 0,Y 333.535,Z 573.185,A -85,B 0,C 180,E1 -14869.383,E2 -14869.383} C_VEL
LIN {X 0,Y 335.238,Z 564.28,A -85,B 0,C 180,E1 -14870.558,E2 -14870.558} C_VEL
LIN {X 0,Y 335.872,Z 553.143,A -85,B 0,C 180,E1 -14871.933,E2 -14871.933} C_VEL
LIN {X 0,Y 335.071,Z 541.555,A -85,B 0,C 180,E1 -14873.328,E2 -14873.328} C_VEL
LIN {X 0,Y 332.849,Z 529.578,A -85,B 0,C 180,E1 -14874.779,E2 -14874.779} C_VEL
LIN {X 0,Y 330.498,Z 520.62,A -85,B 0,C 180,E1 -14875.895,E2 -14875.895} C_VEL
LIN {X 0,Y 328.389,Z 514.694,A -85,B 0,C 180,E1 -14876.707,E2 -14876.707} C_VEL
LIN {X 0,Y 327.324,Z 510.93,A -85,B 0,C 180,E1 -14877.168,E2 -14877.168} C_VEL
LIN {X 0,Y 328.422,Z 504.938,A -85,B 0,C 180,E1 -14881.133,E2 -14881.133} C_VEL
LIN {X 0,Y 329.194,Z 501.459,A -85,B 0,C 180,E1 -14883.716,E2 -14883.716} C_VEL
LIN {X 0,Y 329.892,Z 498.013,A -85,B 0,C 180,E1 -14886.621,E2 -14886.621} C_VEL
LIN {X 0,Y 330.01,Z 496.448,A -85,B 0,C 180,E1 -14888.141,E2 -14888.141} C_VEL
LIN {X 0,Y 329.891,Z 494.849,A -85,B 0,C 180,E1 -14889.92,E2 -14889.92} C_VEL
LIN {X 0,Y 329.559,Z 492.228,A -85,B 0,C 180,E1 -14893.526,E2 -14893.526} C_VEL
LIN {X 0,Y 329.221,Z 490.494,A -85,B 0,C 180,E1 -14896.912,E2 -14896.912} C_VEL
LIN {X 0,Y 328.934,Z 489.424,A -85,B 0,C 180,E1 -14900.28,E2 -14900.28} C_VEL
LIN {X 0,Y 328.704,Z 488.991,A -85,B 0,C 180,E1 -14903.226,E2 -14903.226} C_VEL
LIN {X 0,Y 328.307,Z 489.046,A -85,B 0,C 180,E1 -14906.602,E2 -14906.602} C_VEL
LIN {X 0,Y 327.951,Z 489.408,A -85,B 0,C 180,E1 -14909.048,E2 -14909.048} C_VEL
LIN {X 0,Y 327.316,Z 490.486,A -85,B 0,C 180,E1 -14913.005,E2 -14913.005} C_VEL
LIN {X 0,Y 327.849,Z 492.242,A -85,B 0,C 180,E1 -14913.245,E2 -14913.245} C_VEL
LIN {X 0,Y 329.8,Z 495.191,A -85,B 0,C 180,E1 -14913.864,E2 -14913.864} C_VEL
LIN {X 0,Y 334.993,Z 506.268,A -85,B 0,C 180,E1 -14915.786,E2 -14915.786} C_VEL
LIN {X 0,Y 338.441,Z 516.1,A -85,B 0,C 180,E1 -14917.358,E2 -14917.358} C_VEL
LIN {X 0,Y 339.826,Z 522.46,A -85,B 0,C 180,E1 -14918.321,E2 -14918.321} C_VEL
LIN {X 0,Y 338.895,Z 528.831,A -85,B 0,C 180,E1 -14919.04,E2 -14919.04} C_VEL
LIN {X 0,Y 336.696,Z 540.149,A -85,B 0,C 180,E1 -14920.49,E2 -14920.49} C_VEL
LIN {X 0,Y 334.655,Z 549.468,A -85,B 0,C 180,E1 -14921.955,E2 -14921.955} C_VEL
LIN {X 0,Y 332.467,Z 558.693,A -85,B 0,C 180,E1 -14923.735,E2 -14923.735} C_VEL
LIN {X 0,Y 330.452,Z 567.356,A -85,B 0,C 180,E1 -14925.843,E2 -14925.843} C_VEL
LIN {X 0,Y 329.09,Z 573.262,A -85,B 0,C 180,E1 -14927.669,E2 -14927.669} C_VEL
LIN {X 0,Y 327.863,Z 578,A -85,B 0,C 180,E1 -14929.502,E2 -14929.502} C_VEL
LIN {X 0,Y 326.901,Z 581.902,A -85,B 0,C 180,E1 -14931.476,E2 -14931.476} C_VEL
LIN {X 0,Y 326.334,Z 583.585,A -85,B 0,C 180,E1 -14932.576,E2 -14932.576} C_VEL
LIN {X 0,Y 325.97,Z 585.047,A -85,B 0,C 180,E1 -14933.812,E2 -14933.812} C_VEL
LIN {X 0,Y 325.901,Z 586.094,A -85,B 0,C 180,E1 -14935.052,E2 -14935.052} C_VEL
LIN {X 0,Y 325.662,Z 586.761,A -85,B 0,C 180,E1 -14936.288,E2 -14936.288} C_VEL
LIN {X 0,Y 325.27,Z 586.859,A -85,B 0,C 180,E1 -14938.762,E2 -14938.762} C_VEL
LIN {X 0,Y 325.185,Z 586.317,A -85,B 0,C 180,E1 -14940,E2 -14940} C_VEL
LIN {X 0,Y 325.141,Z 585.346,A -85,B 0,C 180,E1 -14941.239,E2 -14941.239} C_VEL
LIN {X 0,Y 325.14,Z 583.944,A -85,B 0,C 180,E1 -14942.478,E2 -14942.478} C_VEL
LIN {X 0,Y 325.266,Z 581.048,A -85,B 0,C 180,E1 -14944.337,E2 -14944.337} C_VEL
LIN {X 0,Y 325.462,Z 577.115,A -85,B 0,C 180,E1 -14946.199,E2 -14946.199} C_VEL
LIN {X 0,Y 325.784,Z 572.042,A -85,B 0,C 180,E1 -14948.061,E2 -14948.061} C_VEL
LIN {X 0,Y 326.288,Z 565.691,A -85,B 0,C 180,E1 -14949.923,E2 -14949.923} C_VEL
LIN {X 0,Y 327.007,Z 557.829,A -85,B 0,C 180,E1 -14951.781,E2 -14951.781} C_VEL
LIN {X 0,Y 327.889,Z 548.049,A -85,B 0,C 180,E1 -14953.638,E2 -14953.638} C_VEL
LIN {X 0,Y 328.862,Z 538.112,A -85,B 0,C 180,E1 -14955.177,E2 -14955.177} C_VEL
LIN {X 0,Y 329.705,Z 527.588,A -85,B 0,C 180,E1 -14956.508,E2 -14956.508} C_VEL
LIN {X 0,Y 330.686,Z 515.021,A -85,B 0,C 180,E1 -14957.789,E2 -14957.789} C_VEL
LIN {X 0,Y 330.929,Z 509.62,A -85,B 0,C 180,E1 -14958.256,E2 -14958.256} C_VEL
LIN {X 0,Y 328.172,Z 496.109,A -85,B 0,C 180,E1 -14959.33,E2 -14959.33} C_VEL
LIN {X 0,Y 325.474,Z 482.705,A -85,B 0,C 180,E1 -14960.149,E2 -14960.149} C_VEL
LIN {X 0,Y 325.351,Z 481.841,A -85,B 0,C 180,E1 -14960.22,E2 -14960.22} C_VEL
LIN {X 0,Y 325.422,Z 478.081,A -85,B 0,C 180,E1 -14964.226,E2 -14964.226} C_VEL
LIN {X 0,Y 325.593,Z 475.932,A -85,B 0,C 180,E1 -14966.955,E2 -14966.955} C_VEL
LIN {X 0,Y 325.986,Z 475.881,A -85,B 0,C 180,E1 -14970.416,E2 -14970.416} C_VEL
LIN {X 0,Y 326.33,Z 475.836,A -85,B 0,C 180,E1 -14974.053,E2 -14974.053} C_VEL
LIN {X 0,Y 326.606,Z 475.798,A -85,B 0,C 180,E1 -14977.233,E2 -14977.233} C_VEL
LIN {X 0,Y 326.594,Z 475.805,A -85,B 0,C 180,E1 -14980.209,E2 -14980.209} C_VEL
LIN {X 0,Y 326.566,Z 475.804,A -85,B 0,C 180,E1 -14983.526,E2 -14983.526} C_VEL
LIN {X 0,Y 326.58,Z 475.802,A -85,B 0,C 180,E1 -14987.028,E2 -14987.028} C_VEL
LIN {X 0,Y 326.616,Z 475.798,A -85,B 0,C 180,E1 -14990.773,E2 -14990.773} C_VEL
LIN {X 0,Y 326.617,Z 475.8,A -85,B 0,C 180,E1 -14994.481,E2 -14994.481} C_VEL
LIN {X 0,Y 326.614,Z 475.798,A -85,B 0,C 180,E1 -14997.456,E2 -14997.456} C_VEL
LIN {X 0,Y 326.665,Z 475.795,A -85,B 0,C 180,E1 -15000.341,E2 -15000.341} C_VEL
LIN {X 0,Y 326.694,Z 475.79,A -85,B 0,C 180,E1 -15004.516,E2 -15004.516} C_VEL
LIN {X 0,Y 326.651,Z 475.795,A -85,B 0,C 180,E1 -15008.546,E2 -15008.546} C_VEL
LIN {X 0,Y 326.749,Z 475.781,A -85,B 0,C 180,E1 -15011.178,E2 -15011.178} C_VEL
LIN {X 0,Y 326.768,Z 475.779,A -85,B 0,C 180,E1 -15015.433,E2 -15015.433} C_VEL
LIN {X 0,Y 326.775,Z 475.778,A -85,B 0,C 180,E1 -15018.839,E2 -15018.839} C_VEL
LIN {X 0,Y 326.985,Z 475.752,A -85,B 0,C 180,E1 -15022.59,E2 -15022.59} C_VEL
LIN {X 0,Y 326.782,Z 475.776,A -85,B 0,C 180,E1 -15025.065,E2 -15025.065} C_VEL
LIN {X 0,Y 327.051,Z 475.745,A -85,B 0,C 180,E1 -15027.537,E2 -15027.537} C_VEL
LIN {X 0,Y 327.202,Z 475.73,A -85,B 0,C 180,E1 -15030,E2 -15030} C_VEL
LIN {X 0,Y 327.05,Z 475.745,A -85,B 0,C 180,E1 -15032.463,E2 -15032.463} C_VEL
LIN {X 0,Y 326.957,Z 475.758,A -85,B 0,C 180,E1 -15036.17,E2 -15036.17} C_VEL
LIN {X 0,Y 326.809,Z 475.779,A -85,B 0,C 180,E1 -15039.906,E2 -15039.906} C_VEL
LIN {X 0,Y 326.764,Z 475.782,A -85,B 0,C 180,E1 -15043.685,E2 -15043.685} C_VEL
LIN {X 0,Y 326.704,Z 475.788,A -85,B 0,C 180,E1 -15047.528,E2 -15047.528} C_VEL
LIN {X 0,Y 326.665,Z 475.794,A -85,B 0,C 180,E1 -15050.135,E2 -15050.135} C_VEL
LIN {X 0,Y 326.654,Z 475.796,A -85,B 0,C 180,E1 -15054.129,E2 -15054.129} C_VEL
LIN {X 0,Y 326.687,Z 475.788,A -85,B 0,C 180,E1 -15056.858,E2 -15056.858} C_VEL
LIN {X 0,Y 326.638,Z 475.795,A -85,B 0,C 180,E1 -15060.61,E2 -15060.61} C_VEL
LIN {X 0,Y 326.612,Z 475.801,A -85,B 0,C 180,E1 -15064.019,E2 -15064.019} C_VEL
LIN {X 0,Y 326.633,Z 475.796,A -85,B 0,C 180,E1 -15067.239,E2 -15067.239} C_VEL
LIN {X 0,Y 326.582,Z 475.802,A -85,B 0,C 180,E1 -15071.131,E2 -15071.131} C_VEL
LIN {X 0,Y 326.531,Z 475.808,A -85,B 0,C 180,E1 -15074.743,E2 -15074.743} C_VEL
LIN {X 0,Y 326.58,Z 475.804,A -85,B 0,C 180,E1 -15078.154,E2 -15078.154} C_VEL
LIN {X 0,Y 326.599,Z 475.802,A -85,B 0,C 180,E1 -15081.387,E2 -15081.387} C_VEL
LIN {X 0,Y 326.536,Z 475.807,A -85,B 0,C 180,E1 -15084.47,E2 -15084.47} C_VEL
LIN {X 0,Y 326.345,Z 475.834,A -85,B 0,C 180,E1 -15087.426,E2 -15087.426} C_VEL
LIN {X 0,Y 325.955,Z 475.88,A -85,B 0,C 180,E1 -15090.27,E2 -15090.27} C_VEL
LIN {X 0,Y 325.608,Z 475.924,A -85,B 0,C 180,E1 -15093.046,E2 -15093.046} C_VEL
LIN {X 0,Y 325.364,Z 476.051,A -85,B 0,C 180,E1 -15095.124,E2 -15095.124} C_VEL
LIN {X 0,Y 325.292,Z 480.498,A -85,B 0,C 180,E1 -15099.302,E2 -15099.302} C_VEL
LIN {X 0,Y 325.274,Z 481.695,A -85,B 0,C 180,E1 -15099.688,E2 -15099.688} C_VEL
LIN {X 0,Y 325.195,Z 484.426,A -85,B 0,C 180,E1 -15100.024,E2 -15100.024} C_VEL
LIN {X 0,Y 324.866,Z 490.615,A -85,B 0,C 180,E1 -15100.395,E2 -15100.395} C_VEL
LIN {X 0,Y 323.283,Z 504.543,A -85,B 0,C 180,E1 -15101.232,E2 -15101.232} C_VEL
LIN {X 0,Y 323.556,Z 509.116,A -85,B 0,C 180,E1 -15101.631,E2 -15101.631} C_VEL
LIN {X 0,Y 323.872,Z 511.29,A -85,B 0,C 180,E1 -15101.824,E2 -15101.824} C_VEL
LIN {X 0,Y 323.04,Z 523.321,A -85,B 0,C 180,E1 -15102.985,E2 -15102.985} C_VEL
LIN {X 0,Y 322.142,Z 534.574,A -85,B 0,C 180,E1 -15104.337,E2 -15104.337} C_VEL
LIN {X 0,Y 321.184,Z 544.195,A -85,B 0,C 180,E1 -15105.749,E2 -15105.749} C_VEL
LIN {X 0,Y 320.109,Z 554.694,A -85,B 0,C 180,E1 -15107.639,E2 -15107.639} C_VEL
LIN {X 0,Y 319.372,Z 563.174,A -85,B 0,C 180,E1 -15109.54,E2 -15109.54} C_VEL
LIN {X 0,Y 318.707,Z 571.072,A -85,B 0,C 180,E1 -15111.759,E2 -15111.759} C_VEL
LIN {X 0,Y 318.364,Z 576.379,A -85,B 0,C 180,E1 -15113.663,E2 -15113.663} C_VEL
LIN {X 0,Y 318.195,Z 580.515,A -85,B 0,C 180,E1 -15115.566,E2 -15115.566} C_VEL
LIN {X 0,Y 318.041,Z 583.596,A -85,B 0,C 180,E1 -15117.467,E2 -15117.467} C_VEL
LIN {X 0,Y 318.006,Z 585.087,A -85,B 0,C 180,E1 -15118.733,E2 -15118.733} C_VEL
LIN {X 0,Y 318.051,Z 586.174,A -85,B 0,C 180,E1 -15120,E2 -15120} C_VEL
LIN {X 0,Y 318.152,Z 586.849,A -85,B 0,C 180,E1 -15121.265,E2 -15121.265} C_VEL
LIN {X 0,Y 318.347,Z 587.079,A -85,B 0,C 180,E1 -15122.53,E2 -15122.53} C_VEL
LIN {X 0,Y 318.573,Z 586.92,A -85,B 0,C 180,E1 -15123.794,E2 -15123.794} C_VEL
LIN {X 0,Y 318.733,Z 586.387,A -85,B 0,C 180,E1 -15125.06,E2 -15125.06} C_VEL
LIN {X 0,Y 318.861,Z 585.436,A -85,B 0,C 180,E1 -15126.327,E2 -15126.327} C_VEL
LIN {X 0,Y 319.958,Z 582.246,A -85,B 0,C 180,E1 -15128.845,E2 -15128.845} C_VEL
LIN {X 0,Y 320.842,Z 578.765,A -85,B 0,C 180,E1 -15130.73,E2 -15130.73} C_VEL
LIN {X 0,Y 322.141,Z 574.197,A -85,B 0,C 180,E1 -15132.601,E2 -15132.601} C_VEL
LIN {X 0,Y 323.589,Z 568.471,A -85,B 0,C 180,E1 -15134.464,E2 -15134.464} C_VEL
LIN {X 0,Y 325.685,Z 560.147,A -85,B 0,C 180,E1 -15136.614,E2 -15136.614} C_VEL
LIN {X 0,Y 327.962,Z 551.233,A -85,B 0,C 180,E1 -15138.426,E2 -15138.426} C_VEL
LIN {X 0,Y 330.383,Z 540.758,A -85,B 0,C 180,E1 -15140.141,E2 -15140.141} C_VEL
LIN {X 0,Y 332.581,Z 530.295,A -85,B 0,C 180,E1 -15141.54,E2 -15141.54} C_VEL
LIN {X 0,Y 333.741,Z 523.869,A -85,B 0,C 180,E1 -15142.275,E2 -15142.275} C_VEL
LIN {X 0,Y 331.709,Z 514.606,A -85,B 0,C 180,E1 -15143.738,E2 -15143.738} C_VEL
LIN {X 0,Y 328.401,Z 505.046,A -85,B 0,C 180,E1 -15145.341,E2 -15145.341} C_VEL
LIN {X 0,Y 324.763,Z 497.163,A -85,B 0,C 180,E1 -15146.794,E2 -15146.794} C_VEL
LIN {X 0,Y 322.749,Z 493.209,A -85,B 0,C 180,E1 -15147.581,E2 -15147.581} C_VEL
LIN {X 0,Y 320.886,Z 490.026,A -85,B 0,C 180,E1 -15148.267,E2 -15148.267} C_VEL
LIN {X 0,Y 320.59,Z 488.994,A -85,B 0,C 180,E1 -15148.477,E2 -15148.477} C_VEL
LIN {X 0,Y 320.947,Z 486.799,A -85,B 0,C 180,E1 -15151.705,E2 -15151.705} C_VEL
LIN {X 0,Y 321.113,Z 485.071,A -85,B 0,C 180,E1 -15154.684,E2 -15154.684} C_VEL
LIN {X 0,Y 321.088,Z 483.612,A -85,B 0,C 180,E1 -15158.003,E2 -15158.003} C_VEL
LIN {X 0,Y 320.987,Z 482.768,A -85,B 0,C 180,E1 -15161.06,E2 -15161.06} C_VEL
LIN {X 0,Y 320.978,Z 482.508,A -85,B 0,C 180,E1 -15164.48,E2 -15164.48} C_VEL
LIN {X 0,Y 320.915,Z 483.032,A -85,B 0,C 180,E1 -15167.242,E2 -15167.242} C_VEL
LIN {X 0,Y 320.943,Z 484.057,A -85,B 0,C 180,E1 -15169.364,E2 -15169.364} C_VEL
LIN {X 0,Y 321.691,Z 488.592,A -85,B 0,C 180,E1 -15172.286,E2 -15172.286} C_VEL
LIN {X 0,Y 321.705,Z 492.444,A -85,B 0,C 180,E1 -15174.649,E2 -15174.649} C_VEL
LIN {X 0,Y 320.821,Z 498.602,A -85,B 0,C 180,E1 -15178.281,E2 -15178.281} C_VEL
LIN {X 0,Y 320.123,Z 504.114,A -85,B 0,C 180,E1 -15181.422,E2 -15181.422} C_VEL
LIN {X 0,Y 320.822,Z 507.866,A -85,B 0,C 180,E1 -15181.865,E2 -15181.865} C_VEL
LIN {X 0,Y 322.053,Z 510.964,A -85,B 0,C 180,E1 -15182.341,E2 -15182.341} C_VEL
LIN {X 0,Y 325.561,Z 524.361,A -85,B 0,C 180,E1 -15184.078,E2 -15184.078} C_VEL
LIN {X 0,Y 327.826,Z 537.105,A -85,B 0,C 180,E1 -15185.66,E2 -15185.66} C_VEL
LIN {X 0,Y 328.871,Z 549.514,A -85,B 0,C 180,E1 -15187.213,E2 -15187.213} C_VEL
LIN {X 0,Y 328.647,Z 559.055,A -85,B 0,C 180,E1 -15188.419,E2 -15188.419} C_VEL
LIN {X 0,Y 327.762,Z 567.754,A -85,B 0,C 180,E1 -15189.608,E2 -15189.608} C_VEL
LIN {X 0,Y 325.559,Z 577.865,A -85,B 0,C 180,E1 -15191.106,E2 -15191.106} C_VEL
LIN {X 0,Y 323.722,Z 586.544,A -85,B 0,C 180,E1 -15192.664,E2 -15192.664} C_VEL
LIN {X 0,Y 321.858,Z 595.061,A -85,B 0,C 180,E1 -15194.504,E2 -15194.504} C_VEL
LIN {X 0,Y 320.469,Z 602.09,A -85,B 0,C 180,E1 -15196.364,E2 -15196.364} C_VEL
LIN {X 0,Y 319.155,Z 608.749,A -85,B 0,C 180,E1 -15198.569,E2 -15198.569} C_VEL
LIN {X 0,Y 318.499,Z 613.259,A -85,B 0,C 180,E1 -15200.474,E2 -15200.474} C_VEL
LIN {X 0,Y 318.092,Z 616.728,A -85,B 0,C 180,E1 -15202.382,E2 -15202.382} C_VEL
LIN {X 0,Y 318.009,Z 618.903,A -85,B 0,C 180,E1 -15203.988,E2 -15203.988} C_VEL
LIN {X 0,Y 317.952,Z 620.768,A -85,B 0,C 180,E1 -15206.198,E2 -15206.198} C_VEL
LIN {X 0,Y 318.174,Z 621.836,A -85,B 0,C 180,E1 -15208.734,E2 -15208.734} C_VEL
LIN {X 0,Y 318.161,Z 622.628,A -85,B 0,C 180,E1 -15210,E2 -15210} C_VEL
LIN {X 0,Y 318.091,Z 622.973,A -85,B 0,C 180,E1 -15211.266,E2 -15211.266} C_VEL
LIN {X 0,Y 317.903,Z 622.366,A -85,B 0,C 180,E1 -15213.803,E2 -15213.803} C_VEL
LIN {X 0,Y 317.859,Z 620.796,A -85,B 0,C 180,E1 -15215.749,E2 -15215.749} C_VEL
LIN {X 0,Y 318.201,Z 617.364,A -85,B 0,C 180,E1 -15218.254,E2 -15218.254} C_VEL
LIN {X 0,Y 318.72,Z 613.588,A -85,B 0,C 180,E1 -15220.161,E2 -15220.161} C_VEL
LIN {X 0,Y 319.455,Z 608.794,A -85,B 0,C 180,E1 -15222.064,E2 -15222.064} C_VEL
LIN {X 0,Y 320.974,Z 601.748,A -85,B 0,C 180,E1 -15224.26,E2 -15224.26} C_VEL
LIN {X 0,Y 322.634,Z 592.943,A -85,B 0,C 180,E1 -15226.45,E2 -15226.45} C_VEL
LIN {X 0,Y 324.804,Z 583.722,A -85,B 0,C 180,E1 -15228.285,E2 -15228.285} C_VEL
LIN {X 0,Y 327.391,Z 572.508,A -85,B 0,C 180,E1 -15230.088,E2 -15230.088} C_VEL
LIN {X 0,Y 328.88,Z 564.803,A -85,B 0,C 180,E1 -15231.138,E2 -15231.138} C_VEL
LIN {X 0,Y 329.665,Z 553.928,A -85,B 0,C 180,E1 -15232.565,E2 -15232.565} C_VEL
LIN {X 0,Y 329,Z 543.141,A -85,B 0,C 180,E1 -15233.946,E2 -15233.946} C_VEL
LIN {X 0,Y 327.004,Z 531.328,A -85,B 0,C 180,E1 -15235.489,E2 -15235.489} C_VEL
LIN {X 0,Y 324.303,Z 521.268,A -85,B 0,C 180,E1 -15236.883,E2 -15236.883} C_VEL
LIN {X 0,Y 322.248,Z 514.888,A -85,B 0,C 180,E1 -15237.805,E2 -15237.805} C_VEL
LIN {X 0,Y 320.86,Z 511.295,A -85,B 0,C 180,E1 -15238.375,E2 -15238.375} C_VEL
LIN {X 0,Y 320.673,Z 509.93,A -85,B 0,C 180,E1 -15238.548,E2 -15238.548} C_VEL
LIN {X 0,Y 321.561,Z 505.554,A -85,B 0,C 180,E1 -15241.637,E2 -15241.637} C_VEL
LIN {X 0,Y 322.396,Z 501.874,A -85,B 0,C 180,E1 -15244.526,E2 -15244.526} C_VEL
LIN {X 0,Y 322.884,Z 499.768,A -85,B 0,C 180,E1 -15246.356,E2 -15246.356} C_VEL
LIN {X 0,Y 323.017,Z 497.058,A -85,B 0,C 180,E1 -15249.121,E2 -15249.121} C_VEL
LIN {X 0,Y 322.705,Z 494.487,A -85,B 0,C 180,E1 -15252.465,E2 -15252.465} C_VEL
LIN {X 0,Y 322.397,Z 492.594,A -85,B 0,C 180,E1 -15255.767,E2 -15255.767} C_VEL
LIN {X 0,Y 322.093,Z 491.311,A -85,B 0,C 180,E1 -15259.111,E2 -15259.111} C_VEL
LIN {X 0,Y 321.879,Z 490.628,A -85,B 0,C 180,E1 -15262.312,E2 -15262.312} C_VEL
LIN {X 0,Y 321.497,Z 490.497,A -85,B 0,C 180,E1 -15265.364,E2 -15265.364} C_VEL
LIN {X 0,Y 321.032,Z 490.811,A -85,B 0,C 180,E1 -15268.626,E2 -15268.626} C_VEL
LIN {X 0,Y 320.61,Z 491.593,A -85,B 0,C 180,E1 -15271.659,E2 -15271.659} C_VEL
LIN {X 0,Y 321.486,Z 493.978,A -85,B 0,C 180,E1 -15272.062,E2 -15272.062} C_VEL
LIN {X 0,Y 323.186,Z 496.506,A -85,B 0,C 180,E1 -15272.673,E2 -15272.673} C_VEL
LIN {X 0,Y 328.137,Z 506.359,A -85,B 0,C 180,E1 -15274.637,E2 -15274.637} C_VEL
LIN {X 0,Y 331.566,Z 515.511,A -85,B 0,C 180,E1 -15276.251,E2 -15276.251} C_VEL
LIN {X 0,Y 333.44,Z 522.701,A -85,B 0,C 180,E1 -15277.447,E2 -15277.447} C_VEL
LIN {X 0,Y 333.896,Z 525.195,A -85,B 0,C 180,E1 -15277.84,E2 -15277.84} C_VEL
LIN {X 0,Y 331.525,Z 536.988,A -85,B 0,C 180,E1 -15279.284,E2 -15279.284} C_VEL
LIN {X 0,Y 329.008,Z 548.16,A -85,B 0,C 180,E1 -15280.989,E2 -15280.989} C_VEL
LIN {X 0,Y 326.576,Z 557.714,A -85,B 0,C 180,E1 -15282.788,E2 -15282.788} C_VEL
LIN {X 0,Y 324.618,Z 565.474,A -85,B 0,C 180,E1 -15284.621,E2 -15284.621} C_VEL
LIN {X 0,Y 322.691,Z 572.729,A -85,B 0,C 180,E1 -15286.781,E2 -15286.781} C_VEL
LIN {X 0,Y 321.255,Z 577.688,A -85,B 0,C 180,E1 -15288.645,E2 -15288.645} C_VEL
LIN {X 0,Y 320.306,Z 581.519,A -85,B 0,C 180,E1 -15290.528,E2 -15290.528} C_VEL
LIN {X 0,Y 319.347,Z 584.394,A -85,B 0,C 180,E1 -15292.413,E2 -15292.413} C_VEL
LIN {X 0,Y 318.945,Z 585.794,A -85,B 0,C 180,E1 -15293.675,E2 -15293.675} C_VEL
LIN {X 0,Y 318.851,Z 586.763,A -85,B 0,C 180,E1 -15294.942,E2 -15294.942} C_VEL
LIN {X 0,Y 318.607,Z 587.321,A -85,B 0,C 180,E1 -15296.206,E2 -15296.206} C_VEL
LIN {X 0,Y 318.198,Z 587.283,A -85,B 0,C 180,E1 -15298.735,E2 -15298.735} C_VEL
LIN {X 0,Y 318.093,Z 586.658,A -85,B 0,C 180,E1 -15300,E2 -15300} C_VEL
LIN {X 0,Y 318.046,Z 585.593,A -85,B 0,C 180,E1 -15301.267,E2 -15301.267} C_VEL
LIN {X 0,Y 318.049,Z 584.125,A -85,B 0,C 180,E1 -15302.533,E2 -15302.533} C_VEL
LIN {X 0,Y 318.204,Z 581.103,A -85,B 0,C 180,E1 -15304.434,E2 -15304.434} C_VEL
LIN {X 0,Y 318.384,Z 577.034,A -85,B 0,C 180,E1 -15306.337,E2 -15306.337} C_VEL
LIN {X 0,Y 318.717,Z 571.813,A -85,B 0,C 180,E1 -15308.241,E2 -15308.241} C_VEL
LIN {X 0,Y 319.275,Z 565.308,A -85,B 0,C 180,E1 -15310.143,E2 -15310.143} C_VEL
LIN {X 0,Y 319.997,Z 557.226,A -85,B 0,C 180,E1 -15312.043,E2 -15312.043} C_VEL
LIN {X 0,Y 320.95,Z 547.296,A -85,B 0,C 180,E1 -15313.938,E2 -15313.938} C_VEL
LIN {X 0,Y 321.993,Z 537.096,A -85,B 0,C 180,E1 -15315.509,E2 -15315.509} C_VEL
LIN {X 0,Y 322.959,Z 525.016,A -85,B 0,C 180,E1 -15317.019,E2 -15317.019} C_VEL
LIN {X 0,Y 323.838,Z 513.306,A -85,B 0,C 180,E1 -15318.178,E2 -15318.178} C_VEL
LIN {X 0,Y 323.979,Z 511.502,A -85,B 0,C 180,E1 -15318.334,E2 -15318.334} C_VEL
LIN {X 0,Y 321.736,Z 499.611,A -85,B 0,C 180,E1 -15319.348,E2 -15319.348} C_VEL
LIN {X 0,Y 318.905,Z 485.439,A -85,B 0,C 180,E1 -15320.274,E2 -15320.274} C_VEL
LIN {X 0,Y 318.28,Z 482.214,A -85,B 0,C 180,E1 -15320.48,E2 -15320.48} C_VEL
LIN {X 0,Y 318.392,Z 478.212,A -85,B 0,C 180,E1 -15324.797,E2 -15324.797} C_VEL
LIN {X 0,Y 318.445,Z 476.95,A -85,B 0,C 180,E1 -15326.193,E2 -15326.193} C_VEL
LIN {X 0,Y 318.775,Z 476.774,A -85,B 0,C 180,E1 -15329.015,E2 -15329.015} C_VEL
LIN {X 0,Y 319.085,Z 476.737,A -85,B 0,C 180,E1 -15331.912,E2 -15331.912} C_VEL
LIN {X 0,Y 319.436,Z 476.692,A -85,B 0,C 180,E1 -15335.506,E2 -15335.506} C_VEL
LIN {X 0,Y 319.533,Z 476.683,A -85,B 0,C 180,E1 -15338.014,E2 -15338.014} C_VEL
LIN {X 0,Y 319.529,Z 476.68,A -85,B 0,C 180,E1 -15341.597,E2 -15341.597} C_VEL
LIN {X 0,Y 319.492,Z 476.684,A -85,B 0,C 180,E1 -15345.258,E2 -15345.258} C_VEL
LIN {X 0,Y 319.532,Z 476.681,A -85,B 0,C 180,E1 -15348.712,E2 -15348.712} C_VEL
LIN {X 0,Y 319.582,Z 476.678,A -85,B 0,C 180,E1 -15352.344,E2 -15352.344} C_VEL
LIN {X 0,Y 319.564,Z 476.675,A -85,B 0,C 180,E1 -15355.124,E2 -15355.124} C_VEL
LIN {X 0,Y 319.575,Z 476.674,A -85,B 0,C 180,E1 -15359.058,E2 -15359.058} C_VEL
LIN {X 0,Y 319.613,Z 476.672,A -85,B 0,C 180,E1 -15362.498,E2 -15362.498} C_VEL
LIN {X 0,Y 319.609,Z 476.67,A -85,B 0,C 180,E1 -15365.304,E2 -15365.304} C_VEL
LIN {X 0,Y 319.601,Z 476.676,A -85,B 0,C 180,E1 -15368.048,E2 -15368.048} C_VEL
LIN {X 0,Y 319.694,Z 476.659,A -85,B 0,C 180,E1 -15370.962,E2 -15370.962} C_VEL
LIN {X 0,Y 319.735,Z 476.654,A -85,B 0,C 180,E1 -15375.276,E2 -15375.276} C_VEL
LIN {X 0,Y 319.763,Z 476.655,A -85,B 0,C 180,E1 -15379.873,E2 -15379.873} C_VEL
LIN {X 0,Y 319.938,Z 476.631,A -85,B 0,C 180,E1 -15382.426,E2 -15382.426} C_VEL
LIN {X 0,Y 319.751,Z 476.652,A -85,B 0,C 180,E1 -15384.956,E2 -15384.956} C_VEL
LIN {X 0,Y 319.995,Z 476.623,A -85,B 0,C 180,E1 -15387.482,E2 -15387.482} C_VEL
LIN {X 0,Y 320.154,Z 476.608,A -85,B 0,C 180,E1 -15390,E2 -15390} C_VEL
LIN {X 0,Y 319.994,Z 476.623,A -85,B 0,C 180,E1 -15392.518,E2 -15392.518} C_VEL
LIN {X 0,Y 319.914,Z 476.634,A -85,B 0,C 180,E1 -15396.306,E2 -15396.306} C_VEL
LIN {X 0,Y 319.756,Z 476.656,A -85,B 0,C 180,E1 -15400.127,E2 -15400.127} C_VEL
LIN {X 0,Y 319.735,Z 476.654,A -85,B 0,C 180,E1 -15404.724,E2 -15404.724} C_VEL
LIN {X 0,Y 319.693,Z 476.659,A -85,B 0,C 180,E1 -15409.038,E2 -15409.038} C_VEL
LIN {X 0,Y 319.566,Z 476.676,A -85,B 0,C 180,E1 -15413.32,E2 -15413.32} C_VEL
LIN {X 0,Y 319.638,Z 476.67,A -85,B 0,C 180,E1 -15416.088,E2 -15416.088} C_VEL
LIN {X 0,Y 319.584,Z 476.673,A -85,B 0,C 180,E1 -15418.934,E2 -15418.934} C_VEL
LIN {X 0,Y 319.536,Z 476.685,A -85,B 0,C 180,E1 -15421.862,E2 -15421.862} C_VEL
LIN {X 0,Y 319.585,Z 476.676,A -85,B 0,C 180,E1 -15425.543,E2 -15425.543} C_VEL
LIN {X 0,Y 319.578,Z 476.677,A -85,B 0,C 180,E1 -15428.008,E2 -15428.008} C_VEL
LIN {X 0,Y 319.529,Z 476.684,A -85,B 0,C 180,E1 -15431.597,E2 -15431.597} C_VEL
LIN {X 0,Y 319.492,Z 476.686,A -85,B 0,C 180,E1 -15435.257,E2 -15435.257} C_VEL
LIN {X 0,Y 319.532,Z 476.679,A -85,B 0,C 180,E1 -15438.712,E2 -15438.712} C_VEL
LIN {X 0,Y 319.548,Z 476.678,A -85,B 0,C 180,E1 -15442.351,E2 -15442.351} C_VEL
LIN {X 0,Y 319.446,Z 476.691,A -85,B 0,C 180,E1 -15445.109,E2 -15445.109} C_VEL
LIN {X 0,Y 319.171,Z 476.726,A -85,B 0,C 180,E1 -15448.097,E2 -15448.097} C_VEL
LIN {X 0,Y 318.802,Z 476.771,A -85,B 0,C 180,E1 -15450.988,E2 -15450.988} C_VEL
LIN {X 0,Y 318.473,Z 476.816,A -85,B 0,C 180,E1 -15453.809,E2 -15453.809} C_VEL
LIN {X 0,Y 318.287,Z 476.95,A -85,B 0,C 180,E1 -15455.368,E2 -15455.368} C_VEL
LIN {X 0,Y 318.253,Z 481.519,A -85,B 0,C 180,E1 -15459.689,E2 -15459.689} C_VEL
LIN {X 0,Y 320.975,Z 495.839,A -85,B 0,C 180,E1 -15460.56,E2 -15460.56} C_VEL
LIN {X 0,Y 323.556,Z 509.116,A -85,B 0,C 180,E1 -15461.631,E2 -15461.631} C_VEL
LIN {X 0,Y 323.69,Z 512.643,A -85,B 0,C 180,E1 -15461.939,E2 -15461.939} C_VEL
LIN {X 0,Y 322.479,Z 517.854,A -85,B 0,C 180,E1 -15462.391,E2 -15462.391} C_VEL
LIN {X 0,Y 316.344,Z 530.812,A -85,B 0,C 180,E1 -15463.689,E2 -15463.689} C_VEL
LIN {X 0,Y 315.011,Z 535.605,A -85,B 0,C 180,E1 -15464.299,E2 -15464.299} C_VEL
LIN {X 0,Y 314.059,Z 545.14,A -85,B 0,C 180,E1 -15465.749,E2 -15465.749} C_VEL
LIN {X 0,Y 313.003,Z 555.569,A -85,B 0,C 180,E1 -15467.683,E2 -15467.683} C_VEL
LIN {X 0,Y 312.26,Z 563.952,A -85,B 0,C 180,E1 -15469.627,E2 -15469.627} C_VEL
LIN {X 0,Y 311.672,Z 570.768,A -85,B 0,C 180,E1 -15471.571,E2 -15471.571} C_VEL
LIN {X 0,Y 311.239,Z 577.111,A -85,B 0,C 180,E1 -15473.875,E2 -15473.875} C_VEL
LIN {X 0,Y 311.052,Z 581.687,A -85,B 0,C 180,E1 -15476.113,E2 -15476.113} C_VEL
LIN {X 0,Y 310.954,Z 583.729,A -85,B 0,C 180,E1 -15477.409,E2 -15477.409} C_VEL
LIN {X 0,Y 310.91,Z 585.299,A -85,B 0,C 180,E1 -15478.704,E2 -15478.704} C_VEL
LIN {X 0,Y 311.063,Z 587.214,A -85,B 0,C 180,E1 -15481.294,E2 -15481.294} C_VEL
LIN {X 0,Y 311.284,Z 587.555,A -85,B 0,C 180,E1 -15482.588,E2 -15482.588} C_VEL
LIN {X 0,Y 311.502,Z 587.462,A -85,B 0,C 180,E1 -15483.881,E2 -15483.881} C_VEL
LIN {X 0,Y 311.84,Z 586.163,A -85,B 0,C 180,E1 -15486.47,E2 -15486.47} C_VEL
LIN {X 0,Y 312.877,Z 583.586,A -85,B 0,C 180,E1 -15488.753,E2 -15488.753} C_VEL
LIN {X 0,Y 313.944,Z 579.82,A -85,B 0,C 180,E1 -15490.969,E2 -15490.969} C_VEL
LIN {X 0,Y 315.32,Z 575.424,A -85,B 0,C 180,E1 -15492.878,E2 -15492.878} C_VEL
LIN {X 0,Y 316.878,Z 569.948,A -85,B 0,C 180,E1 -15494.777,E2 -15494.777} C_VEL
LIN {X 0,Y 318.768,Z 563.186,A -85,B 0,C 180,E1 -15496.655,E2 -15496.655} C_VEL
LIN {X 0,Y 321.051,Z 554.878,A -85,B 0,C 180,E1 -15498.506,E2 -15498.506} C_VEL
LIN {X 0,Y 323.716,Z 544.773,A -85,B 0,C 180,E1 -15500.326,E2 -15500.326} C_VEL
LIN {X 0,Y 326.133,Z 534.127,A -85,B 0,C 180,E1 -15501.868,E2 -15501.868} C_VEL
LIN {X 0,Y 327.796,Z 526.546,A -85,B 0,C 180,E1 -15502.79,E2 -15502.79} C_VEL
LIN {X 0,Y 326.693,Z 520.19,A -85,B 0,C 180,E1 -15503.851,E2 -15503.851} C_VEL
LIN {X 0,Y 323.943,Z 510.871,A -85,B 0,C 180,E1 -15505.507,E2 -15505.507} C_VEL
LIN {X 0,Y 320.282,Z 502.102,A -85,B 0,C 180,E1 -15507.226,E2 -15507.226} C_VEL
LIN {X 0,Y 316.52,Z 494.562,A -85,B 0,C 180,E1 -15508.863,E2 -15508.863} C_VEL
LIN {X 0,Y 314.884,Z 492.441,A -85,B 0,C 180,E1 -15509.488,E2 -15509.488} C_VEL
LIN {X 0,Y 313.926,Z 489.909,A -85,B 0,C 180,E1 -15510.042,E2 -15510.042} C_VEL
LIN {X 0,Y 314.216,Z 488.433,A -85,B 0,C 180,E1 -15512.466,E2 -15512.466} C_VEL
LIN {X 0,Y 314.383,Z 486.897,A -85,B 0,C 180,E1 -15515.537,E2 -15515.537} C_VEL
LIN {X 0,Y 314.367,Z 485.758,A -85,B 0,C 180,E1 -15518.753,E2 -15518.753} C_VEL
LIN {X 0,Y 314.376,Z 485.178,A -85,B 0,C 180,E1 -15522.118,E2 -15522.118} C_VEL
LIN {X 0,Y 314.422,Z 485.411,A -85,B 0,C 180,E1 -15525.665,E2 -15525.665} C_VEL
LIN {X 0,Y 314.391,Z 486.157,A -85,B 0,C 180,E1 -15527.884,E2 -15527.884} C_VEL
LIN {X 0,Y 314.434,Z 487.079,A -85,B 0,C 180,E1 -15529.595,E2 -15529.595} C_VEL
LIN {X 0,Y 314.583,Z 489.037,A -85,B 0,C 180,E1 -15532.011,E2 -15532.011} C_VEL
LIN {X 0,Y 314.759,Z 491.362,A -85,B 0,C 180,E1 -15533.496,E2 -15533.496} C_VEL
LIN {X 0,Y 314.305,Z 495.465,A -85,B 0,C 180,E1 -15536.012,E2 -15536.012} C_VEL
LIN {X 0,Y 313.545,Z 500.48,A -85,B 0,C 180,E1 -15538.966,E2 -15538.966} C_VEL
LIN {X 0,Y 313.484,Z 502.644,A -85,B 0,C 180,E1 -15539.777,E2 -15539.777} C_VEL
LIN {X 0,Y 314.569,Z 506.597,A -85,B 0,C 180,E1 -15540.393,E2 -15540.393} C_VEL
LIN {X 0,Y 315.596,Z 509.048,A -85,B 0,C 180,E1 -15540.839,E2 -15540.839} C_VEL
LIN {X 0,Y 316.846,Z 513.652,A -85,B 0,C 180,E1 -15541.504,E2 -15541.504} C_VEL
LIN {X 0,Y 318.908,Z 521.65,A -85,B 0,C 180,E1 -15542.65,E2 -15542.65} C_VEL
LIN {X 0,Y 321.177,Z 533.164,A -85,B 0,C 180,E1 -15544.225,E2 -15544.225} C_VEL
LIN {X 0,Y 322.54,Z 545.494,A -85,B 0,C 180,E1 -15545.867,E2 -15545.867} C_VEL
LIN {X 0,Y 322.785,Z 554.9,A -85,B 0,C 180,E1 -15547.129,E2 -15547.129} C_VEL
LIN {X 0,Y 321.716,Z 567.312,A -85,B 0,C 180,E1 -15548.872,E2 -15548.872} C_VEL
LIN {X 0,Y 319.376,Z 577.315,A -85,B 0,C 180,E1 -15550.392,E2 -15550.392} C_VEL
LIN {X 0,Y 317.02,Z 587.484,A -85,B 0,C 180,E1 -15552.286,E2 -15552.286} C_VEL
LIN {X 0,Y 315.286,Z 594.65,A -85,B 0,C 180,E1 -15553.894,E2 -15553.894} C_VEL
LIN {X 0,Y 313.596,Z 602.455,A -85,B 0,C 180,E1 -15556.059,E2 -15556.059} C_VEL
LIN {X 0,Y 312.167,Z 608.961,A -85,B 0,C 180,E1 -15558.31,E2 -15558.31} C_VEL
LIN {X 0,Y 311.459,Z 613.298,A -85,B 0,C 180,E1 -15560.257,E2 -15560.257} C_VEL
LIN {X 0,Y 311.027,Z 616.619,A -85,B 0,C 180,E1 -15562.208,E2 -15562.208} C_VEL
LIN {X 0,Y 310.901,Z 618.886,A -85,B 0,C 180,E1 -15564.061,E2 -15564.061} C_VEL
LIN {X 0,Y 310.877,Z 620.414,A -85,B 0,C 180,E1 -15566.111,E2 -15566.111} C_VEL
LIN {X 0,Y 311.113,Z 621.186,A -85,B 0,C 180,E1 -15568.706,E2 -15568.706} C_VEL
LIN {X 0,Y 311.104,Z 622.035,A -85,B 0,C 180,E1 -15570,E2 -15570} C_VEL
LIN {X 0,Y 311.013,Z 622.46,A -85,B 0,C 180,E1 -15571.295,E2 -15571.295} C_VEL
LIN {X 0,Y 310.817,Z 622.44,A -85,B 0,C 180,E1 -15572.592,E2 -15572.592} C_VEL
LIN {X 0,Y 310.828,Z 621.999,A -85,B 0,C 180,E1 -15573.889,E2 -15573.889} C_VEL
LIN {X 0,Y 310.828,Z 619.91,A -85,B 0,C 180,E1 -15576.491,E2 -15576.491} C_VEL
LIN {X 0,Y 311.145,Z 617.237,A -85,B 0,C 180,E1 -15578.443,E2 -15578.443} C_VEL
LIN {X 0,Y 311.692,Z 613.625,A -85,B 0,C 180,E1 -15580.392,E2 -15580.392} C_VEL
LIN {X 0,Y 312.507,Z 608.986,A -85,B 0,C 180,E1 -15582.336,E2 -15582.336} C_VEL
LIN {X 0,Y 314.116,Z 602.175,A -85,B 0,C 180,E1 -15584.579,E2 -15584.579} C_VEL
LIN {X 0,Y 315.683,Z 594.624,A -85,B 0,C 180,E1 -15586.589,E2 -15586.589} C_VEL
LIN {X 0,Y 318.143,Z 584.752,A -85,B 0,C 180,E1 -15588.682,E2 -15588.682} C_VEL
LIN {X 0,Y 320.848,Z 573.971,A -85,B 0,C 180,E1 -15590.516,E2 -15590.516} C_VEL
LIN {X 0,Y 322.63,Z 565.575,A -85,B 0,C 180,E1 -15591.735,E2 -15591.735} C_VEL
LIN {X 0,Y 323.464,Z 556.211,A -85,B 0,C 180,E1 -15593.023,E2 -15593.023} C_VEL
LIN {X 0,Y 323.152,Z 546.184,A -85,B 0,C 180,E1 -15594.407,E2 -15594.407} C_VEL
LIN {X 0,Y 321.626,Z 535.406,A -85,B 0,C 180,E1 -15595.915,E2 -15595.915} C_VEL
LIN {X 0,Y 319.324,Z 525.565,A -85,B 0,C 180,E1 -15597.363,E2 -15597.363} C_VEL
LIN {X 0,Y 315.8,Z 514.264,A -85,B 0,C 180,E1 -15599.18,E2 -15599.18} C_VEL
LIN {X 0,Y 314.3,Z 510.496,A -85,B 0,C 180,E1 -15599.876,E2 -15599.876} C_VEL
LIN {X 0,Y 314.079,Z 508.92,A -85,B 0,C 180,E1 -15600.128,E2 -15600.128} C_VEL
LIN {X 0,Y 314.766,Z 505.896,A -85,B 0,C 180,E1 -15602.403,E2 -15602.403} C_VEL
LIN {X 0,Y 315.641,Z 502.317,A -85,B 0,C 180,E1 -15605.374,E2 -15605.374} C_VEL
LIN {X 0,Y 315.969,Z 500.66,A -85,B 0,C 180,E1 -15606.91,E2 -15606.91} C_VEL
LIN {X 0,Y 316.111,Z 498.758,A -85,B 0,C 180,E1 -15608.909,E2 -15608.909} C_VEL
LIN {X 0,Y 315.819,Z 496.457,A -85,B 0,C 180,E1 -15611.882,E2 -15611.882} C_VEL
LIN {X 0,Y 315.492,Z 494.335,A -85,B 0,C 180,E1 -15615.467,E2 -15615.467} C_VEL
LIN {X 0,Y 315.168,Z 492.842,A -85,B 0,C 180,E1 -15619.304,E2 -15619.304} C_VEL
LIN {X 0,Y 314.859,Z 492.135,A -85,B 0,C 180,E1 -15622.939,E2 -15622.939} C_VEL
LIN {X 0,Y 314.521,Z 492.04,A -85,B 0,C 180,E1 -15626.039,E2 -15626.039} C_VEL
LIN {X 0,Y 313.858,Z 492.559,A -85,B 0,C 180,E1 -15630.053,E2 -15630.053} C_VEL
LIN {X 0,Y 314.841,Z 495.216,A -85,B 0,C 180,E1 -15630.588,E2 -15630.588} C_VEL
LIN {X 0,Y 316.556,Z 497.167,A -85,B 0,C 180,E1 -15631.235,E2 -15631.235} C_VEL
LIN {X 0,Y 317.121,Z 498.734,A -85,B 0,C 180,E1 -15631.544,E2 -15631.544} C_VEL
LIN {X 0,Y 321.77,Z 507.645,A -85,B 0,C 180,E1 -15633.574,E2 -15633.574} C_VEL
LIN {X 0,Y 325.082,Z 516.081,A -85,B 0,C 180,E1 -15635.232,E2 -15635.232} C_VEL
LIN {X 0,Y 327.405,Z 524.341,A -85,B 0,C 180,E1 -15636.731,E2 -15636.731} C_VEL
LIN {X 0,Y 327.922,Z 527.739,A -85,B 0,C 180,E1 -15637.308,E2 -15637.308} C_VEL
LIN {X 0,Y 325.105,Z 540.3,A -85,B 0,C 180,E1 -15638.937,E2 -15638.937} C_VEL
LIN {X 0,Y 322.565,Z 550.471,A -85,B 0,C 180,E1 -15640.594,E2 -15640.594} C_VEL
LIN {X 0,Y 320.026,Z 559.598,A -85,B 0,C 180,E1 -15642.425,E2 -15642.425} C_VEL
LIN {X 0,Y 317.972,Z 567.078,A -85,B 0,C 180,E1 -15644.291,E2 -15644.291} C_VEL
LIN {X 0,Y 315.923,Z 574.094,A -85,B 0,C 180,E1 -15646.492,E2 -15646.492} C_VEL
LIN {X 0,Y 314.417,Z 578.839,A -85,B 0,C 180,E1 -15648.395,E2 -15648.395} C_VEL
LIN {X 0,Y 313.378,Z 582.528,A -85,B 0,C 180,E1 -15650.317,E2 -15650.317} C_VEL
LIN {X 0,Y 312.378,Z 585.25,A -85,B 0,C 180,E1 -15652.242,E2 -15652.242} C_VEL
LIN {X 0,Y 311.924,Z 586.549,A -85,B 0,C 180,E1 -15653.532,E2 -15653.532} C_VEL
LIN {X 0,Y 311.805,Z 587.389,A -85,B 0,C 180,E1 -15654.828,E2 -15654.828} C_VEL
LIN {X 0,Y 311.554,Z 587.878,A -85,B 0,C 180,E1 -15656.12,E2 -15656.12} C_VEL
LIN {X 0,Y 311.294,Z 587.987,A -85,B 0,C 180,E1 -15657.412,E2 -15657.412} C_VEL
LIN {X 0,Y 311.111,Z 587.688,A -85,B 0,C 180,E1 -15658.706,E2 -15658.706} C_VEL
LIN {X 0,Y 311,Z 586.95,A -85,B 0,C 180,E1 -15660,E2 -15660} C_VEL
LIN {X 0,Y 310.95,Z 585.818,A -85,B 0,C 180,E1 -15661.295,E2 -15661.295} C_VEL
LIN {X 0,Y 310.962,Z 584.285,A -85,B 0,C 180,E1 -15662.591,E2 -15662.591} C_VEL
LIN {X 0,Y 311.122,Z 581.144,A -85,B 0,C 180,E1 -15664.535,E2 -15664.535} C_VEL
LIN {X 0,Y 311.364,Z 576.385,A -85,B 0,C 180,E1 -15666.707,E2 -15666.707} C_VEL
LIN {X 0,Y 311.761,Z 570.529,A -85,B 0,C 180,E1 -15668.753,E2 -15668.753} C_VEL
LIN {X 0,Y 312.343,Z 563.582,A -85,B 0,C 180,E1 -15670.698,E2 -15670.698} C_VEL
LIN {X 0,Y 313.128,Z 555.042,A -85,B 0,C 180,E1 -15672.641,E2 -15672.641} C_VEL
LIN {X 0,Y 314.214,Z 544.423,A -85,B 0,C 180,E1 -15674.574,E2 -15674.574} C_VEL
LIN {X 0,Y 315.249,Z 534.07,A -85,B 0,C 180,E1 -15676.107,E2 -15676.107} C_VEL
LIN {X 0,Y 316.134,Z 522.779,A -85,B 0,C 180,E1 -15677.465,E2 -15677.465} C_VEL
LIN {X 0,Y 316.881,Z 513.069,A -85,B 0,C 180,E1 -15678.424,E2 -15678.424} C_VEL
LIN {X 0,Y 315.992,Z 506.974,A -85,B 0,C 180,E1 -15678.983,E2 -15678.983} C_VEL
LIN {X 0,Y 313.619,Z 494.814,A -85,B 0,C 180,E1 -15679.949,E2 -15679.949} C_VEL
LIN {X 0,Y 311.208,Z 482.619,A -85,B 0,C 180,E1 -15680.705,E2 -15680.705} C_VEL
LIN {X 0,Y 311.243,Z 479.61,A -85,B 0,C 180,E1 -15683.982,E2 -15683.982} C_VEL
LIN {X 0,Y 311.36,Z 478.273,A -85,B 0,C 180,E1 -15685.46,E2 -15685.46} C_VEL
LIN {X 0,Y 311.475,Z 477.69,A -85,B 0,C 180,E1 -15686.826,E2 -15686.826} C_VEL
LIN {X 0,Y 311.797,Z 477.644,A -85,B 0,C 180,E1 -15689.729,E2 -15689.729} C_VEL
LIN {X 0,Y 312.089,Z 477.608,A -85,B 0,C 180,E1 -15692.716,E2 -15692.716} C_VEL
LIN {X 0,Y 312.428,Z 477.567,A -85,B 0,C 180,E1 -15695.922,E2 -15695.922} C_VEL
LIN {X 0,Y 312.479,Z 477.558,A -85,B 0,C 180,E1 -15699.032,E2 -15699.032} C_VEL
LIN {X 0,Y 312.494,Z 477.56,A -85,B 0,C 180,E1 -15702.432,E2 -15702.432} C_VEL
LIN {X 0,Y 312.462,Z 477.564,A -85,B 0,C 180,E1 -15706.035,E2 -15706.035} C_VEL
LIN {X 0,Y 312.507,Z 477.557,A -85,B 0,C 180,E1 -15709.875,E2 -15709.875} C_VEL
LIN {X 0,Y 312.542,Z 477.552,A -85,B 0,C 180,E1 -15712.617,E2 -15712.617} C_VEL
LIN {X 0,Y 312.523,Z 477.557,A -85,B 0,C 180,E1 -15716.311,E2 -15716.311} C_VEL
LIN {X 0,Y 312.549,Z 477.553,A -85,B 0,C 180,E1 -15720.35,E2 -15720.35} C_VEL
LIN {X 0,Y 312.607,Z 477.547,A -85,B 0,C 180,E1 -15724.064,E2 -15724.064} C_VEL
LIN {X 0,Y 312.592,Z 477.545,A -85,B 0,C 180,E1 -15727.529,E2 -15727.529} C_VEL
LIN {X 0,Y 312.643,Z 477.539,A -85,B 0,C 180,E1 -15731.657,E2 -15731.657} C_VEL
LIN {X 0,Y 312.698,Z 477.533,A -85,B 0,C 180,E1 -15735.686,E2 -15735.686} C_VEL
LIN {X 0,Y 312.707,Z 477.532,A -85,B 0,C 180,E1 -15739.642,E2 -15739.642} C_VEL
LIN {X 0,Y 312.877,Z 477.512,A -85,B 0,C 180,E1 -15742.254,E2 -15742.254} C_VEL
LIN {X 0,Y 312.722,Z 477.528,A -85,B 0,C 180,E1 -15744.842,E2 -15744.842} C_VEL
LIN {X 0,Y 312.994,Z 477.494,A -85,B 0,C 180,E1 -15748.713,E2 -15748.713} C_VEL
LIN {X 0,Y 312.994,Z 477.495,A -85,B 0,C 180,E1 -15751.287,E2 -15751.287} C_VEL
LIN {X 0,Y 312.711,Z 477.529,A -85,B 0,C 180,E1 -15755.158,E2 -15755.158} C_VEL
LIN {X 0,Y 312.822,Z 477.519,A -85,B 0,C 180,E1 -15757.747,E2 -15757.747} C_VEL
LIN {X 0,Y 312.674,Z 477.537,A -85,B 0,C 180,E1 -15761.671,E2 -15761.671} C_VEL
LIN {X 0,Y 312.705,Z 477.53,A -85,B 0,C 180,E1 -15764.888,E2 -15764.888} C_VEL
LIN {X 0,Y 312.634,Z 477.539,A -85,B 0,C 180,E1 -15769.236,E2 -15769.236} C_VEL
LIN {X 0,Y 312.532,Z 477.551,A -85,B 0,C 180,E1 -15772.781,E2 -15772.781} C_VEL
LIN {X 0,Y 312.606,Z 477.547,A -85,B 0,C 180,E1 -15775.935,E2 -15775.935} C_VEL
LIN {X 0,Y 312.542,Z 477.554,A -85,B 0,C 180,E1 -15779.65,E2 -15779.65} C_VEL
LIN {X 0,Y 312.523,Z 477.557,A -85,B 0,C 180,E1 -15783.689,E2 -15783.689} C_VEL
LIN {X 0,Y 312.542,Z 477.552,A -85,B 0,C 180,E1 -15787.383,E2 -15787.383} C_VEL
LIN {X 0,Y 312.494,Z 477.556,A -85,B 0,C 180,E1 -15790.709,E2 -15790.709} C_VEL
LIN {X 0,Y 312.455,Z 477.563,A -85,B 0,C 180,E1 -15794.209,E2 -15794.209} C_VEL
LIN {X 0,Y 312.488,Z 477.561,A -85,B 0,C 180,E1 -15797.918,E2 -15797.918} C_VEL
LIN {X 0,Y 312.499,Z 477.556,A -85,B 0,C 180,E1 -15800.971,E2 -15800.971} C_VEL
LIN {X 0,Y 312.46,Z 477.562,A -85,B 0,C 180,E1 -15804.21,E2 -15804.21} C_VEL
LIN {X 0,Y 312.209,Z 477.594,A -85,B 0,C 180,E1 -15807.298,E2 -15807.298} C_VEL
LIN {X 0,Y 311.871,Z 477.635,A -85,B 0,C 180,E1 -15810.279,E2 -15810.279} C_VEL
LIN {X 0,Y 311.514,Z 477.68,A -85,B 0,C 180,E1 -15813.178,E2 -15813.178} C_VEL
LIN {X 0,Y 311.203,Z 477.91,A -85,B 0,C 180,E1 -15815.66,E2 -15815.66} C_VEL
LIN {X 0,Y 311.176,Z 482.109,A -85,B 0,C 180,E1 -15819.465,E2 -15819.465} C_VEL
LIN {X 0,Y 313.622,Z 494.953,A -85,B 0,C 180,E1 -15820.252,E2 -15820.252} C_VEL
LIN {X 0,Y 316.021,Z 507.43,A -85,B 0,C 180,E1 -15821.242,E2 -15821.242} C_VEL
LIN {X 0,Y 316.759,Z 511.268,A -85,B 0,C 180,E1 -15821.596,E2 -15821.596} C_VEL
LIN {X 0,Y 316.159,Z 521.678,A -85,B 0,C 180,E1 -15822.603,E2 -15822.603} C_VEL
LIN {X 0,Y 315.229,Z 533.394,A -85,B 0,C 180,E1 -15824.004,E2 -15824.004} C_VEL
LIN {X 0,Y 315.011,Z 535.605,A -85,B 0,C 180,E1 -15824.299,E2 -15824.299} C_VEL
LIN {X 0,Y 313.823,Z 540.231,A -85,B 0,C 180,E1 -15824.936,E2 -15824.936} C_VEL
LIN {X 0,Y 310.228,Z 547.348,A -85,B 0,C 180,E1 -15826.022,E2 -15826.022} C_VEL
LIN {X 0,Y 306.75,Z 553.981,A -85,B 0,C 180,E1 -15827.23,E2 -15827.23} C_VEL
LIN {X 0,Y 305.757,Z 557.845,A -85,B 0,C 180,E1 -15828.046,E2 -15828.046} C_VEL
LIN {X 0,Y 305.014,Z 565.954,A -85,B 0,C 180,E1 -15830.048,E2 -15830.048} C_VEL
LIN {X 0,Y 304.457,Z 572.44,A -85,B 0,C 180,E1 -15832.038,E2 -15832.038} C_VEL
LIN {X 0,Y 304.131,Z 577.432,A -85,B 0,C 180,E1 -15833.942,E2 -15833.942} C_VEL
LIN {X 0,Y 303.986,Z 581.68,A -85,B 0,C 180,E1 -15836.023,E2 -15836.023} C_VEL
LIN {X 0,Y 303.871,Z 583.798,A -85,B 0,C 180,E1 -15837.348,E2 -15837.348} C_VEL
LIN {X 0,Y 303.817,Z 585.497,A -85,B 0,C 180,E1 -15838.674,E2 -15838.674} C_VEL
LIN {X 0,Y 303.863,Z 586.727,A -85,B 0,C 180,E1 -15840,E2 -15840} C_VEL
LIN {X 0,Y 304.204,Z 587.994,A -85,B 0,C 180,E1 -15842.648,E2 -15842.648} C_VEL
LIN {X 0,Y 304.432,Z 588.016,A -85,B 0,C 180,E1 -15843.971,E2 -15843.971} C_VEL
LIN {X 0,Y 304.824,Z 586.866,A -85,B 0,C 180,E1 -15846.619,E2 -15846.619} C_VEL
LIN {X 0,Y 305.946,Z 584.46,A -85,B 0,C 180,E1 -15848.969,E2 -15848.969} C_VEL
LIN {X 0,Y 307.072,Z 580.924,A -85,B 0,C 180,E1 -15851.218,E2 -15851.218} C_VEL
LIN {X 0,Y 308.534,Z 576.728,A -85,B 0,C 180,E1 -15853.167,E2 -15853.167} C_VEL
LIN {X 0,Y 310.47,Z 570.425,A -85,B 0,C 180,E1 -15855.425,E2 -15855.425} C_VEL
LIN {X 0,Y 312.922,Z 562.467,A -85,B 0,C 180,E1 -15857.65,E2 -15857.65} C_VEL
LIN {X 0,Y 315.478,Z 553.956,A -85,B 0,C 180,E1 -15859.521,E2 -15859.521} C_VEL
LIN {X 0,Y 318.303,Z 543.57,A -85,B 0,C 180,E1 -15861.365,E2 -15861.365} C_VEL
LIN {X 0,Y 321.014,Z 532.86,A -85,B 0,C 180,E1 -15862.9,E2 -15862.9} C_VEL
LIN {X 0,Y 321.94,Z 528.951,A -85,B 0,C 180,E1 -15863.376,E2 -15863.376} C_VEL
LIN {X 0,Y 320.315,Z 520.236,A -85,B 0,C 180,E1 -15864.964,E2 -15864.964} C_VEL
LIN {X 0,Y 317.199,Z 510.464,A -85,B 0,C 180,E1 -15866.9,E2 -15866.9} C_VEL
LIN {X 0,Y 312.482,Z 499.961,A -85,B 0,C 180,E1 -15869.286,E2 -15869.286} C_VEL
LIN {X 0,Y 310.855,Z 497.61,A -85,B 0,C 180,E1 -15869.988,E2 -15869.988} C_VEL
LIN {X 0,Y 309.938,Z 495.5,A -85,B 0,C 180,E1 -15870.495,E2 -15870.495} C_VEL
LIN {X 0,Y 308.439,Z 493.593,A -85,B 0,C 180,E1 -15871.162,E2 -15871.162} C_VEL
LIN {X 0,Y 307.412,Z 490.909,A -85,B 0,C 180,E1 -15871.863,E2 -15871.863} C_VEL
LIN {X 0,Y 307.605,Z 489.484,A -85,B 0,C 180,E1 -15874.833,E2 -15874.833} C_VEL
LIN {X 0,Y 307.72,Z 488.677,A -85,B 0,C 180,E1 -15876.93,E2 -15876.93} C_VEL
LIN {X 0,Y 307.701,Z 488.012,A -85,B 0,C 180,E1 -15879.757,E2 -15879.757} C_VEL
LIN {X 0,Y 307.794,Z 487.837,A -85,B 0,C 180,E1 -15883.236,E2 -15883.236} C_VEL
LIN {X 0,Y 307.853,Z 488.069,A -85,B 0,C 180,E1 -15885.048,E2 -15885.048} C_VEL
LIN {X 0,Y 307.901,Z 488.656,A -85,B 0,C 180,E1 -15886.921,E2 -15886.921} C_VEL
LIN {X 0,Y 307.936,Z 489.624,A -85,B 0,C 180,E1 -15888.865,E2 -15888.865} C_VEL
LIN {X 0,Y 308.168,Z 492.065,A -85,B 0,C 180,E1 -15891.993,E2 -15891.993} C_VEL
LIN {X 0,Y 308.037,Z 493.988,A -85,B 0,C 180,E1 -15893.615,E2 -15893.615} C_VEL
LIN {X 0,Y 307.553,Z 497.695,A -85,B 0,C 180,E1 -15895.954,E2 -15895.954} C_VEL
LIN {X 0,Y 307.312,Z 501.982,A -85,B 0,C 180,E1 -15898.047,E2 -15898.047} C_VEL
LIN {X 0,Y 309.335,Z 507.776,A -85,B 0,C 180,E1 -15899.204,E2 -15899.204} C_VEL
LIN {X 0,Y 311.412,Z 514.958,A -85,B 0,C 180,E1 -15900.417,E2 -15900.417} C_VEL
LIN {X 0,Y 313.767,Z 524.614,A -85,B 0,C 180,E1 -15901.941,E2 -15901.941} C_VEL
LIN {X 0,Y 315.833,Z 537.581,A -85,B 0,C 180,E1 -15903.831,E2 -15903.831} C_VEL
LIN {X 0,Y 316.761,Z 550.638,A -85,B 0,C 180,E1 -15905.694,E2 -15905.694} C_VEL
LIN {X 0,Y 316.331,Z 560.575,A -85,B 0,C 180,E1 -15907.12,E2 -15907.12} C_VEL
LIN {X 0,Y 315.037,Z 570.159,A -85,B 0,C 180,E1 -15908.574,E2 -15908.574} C_VEL
LIN {X 0,Y 312.377,Z 580.402,A -85,B 0,C 180,E1 -15910.277,E2 -15910.277} C_VEL
LIN {X 0,Y 309.942,Z 590.021,A -85,B 0,C 180,E1 -15912.243,E2 -15912.243} C_VEL
LIN {X 0,Y 307.997,Z 597.482,A -85,B 0,C 180,E1 -15914.108,E2 -15914.108} C_VEL
LIN {X 0,Y 306.454,Z 603.904,A -85,B 0,C 180,E1 -15916.066,E2 -15916.066} C_VEL
LIN {X 0,Y 305.188,Z 609.142,A -85,B 0,C 180,E1 -15918.038,E2 -15918.038} C_VEL
LIN {X 0,Y 304.243,Z 614.495,A -85,B 0,C 180,E1 -15920.694,E2 -15920.694} C_VEL
LIN {X 0,Y 303.982,Z 616.519,A -85,B 0,C 180,E1 -15922.026,E2 -15922.026} C_VEL
LIN {X 0,Y 303.768,Z 619.276,A -85,B 0,C 180,E1 -15924.69,E2 -15924.69} C_VEL
LIN {X 0,Y 303.782,Z 620.066,A -85,B 0,C 180,E1 -15926.02,E2 -15926.02} C_VEL
LIN {X 0,Y 304.052,Z 620.517,A -85,B 0,C 180,E1 -15928.676,E2 -15928.676} C_VEL
LIN {X 0,Y 304.049,Z 621.423,A -85,B 0,C 180,E1 -15930,E2 -15930} C_VEL
LIN {X 0,Y 303.937,Z 621.908,A -85,B 0,C 180,E1 -15931.325,E2 -15931.325} C_VEL
LIN {X 0,Y 303.735,Z 621.979,A -85,B 0,C 180,E1 -15932.652,E2 -15932.652} C_VEL
LIN {X 0,Y 303.732,Z 621.632,A -85,B 0,C 180,E1 -15933.98,E2 -15933.98} C_VEL
LIN {X 0,Y 303.741,Z 619.672,A -85,B 0,C 180,E1 -15936.643,E2 -15936.643} C_VEL
LIN {X 0,Y 303.951,Z 618.107,A -85,B 0,C 180,E1 -15937.975,E2 -15937.975} C_VEL
LIN {X 0,Y 304.445,Z 614.947,A -85,B 0,C 180,E1 -15939.97,E2 -15939.97} C_VEL
LIN {X 0,Y 305.208,Z 610.796,A -85,B 0,C 180,E1 -15941.961,E2 -15941.961} C_VEL
LIN {X 0,Y 306.483,Z 605.644,A -85,B 0,C 180,E1 -15943.932,E2 -15943.932} C_VEL
LIN {X 0,Y 308.26,Z 598.181,A -85,B 0,C 180,E1 -15946.218,E2 -15946.218} C_VEL
LIN {X 0,Y 310.436,Z 589.915,A -85,B 0,C 180,E1 -15948.231,E2 -15948.231} C_VEL
LIN {X 0,Y 312.887,Z 580.916,A -85,B 0,C 180,E1 -15950.032,E2 -15950.032} C_VEL
LIN {X 0,Y 315.653,Z 570.543,A -85,B 0,C 180,E1 -15951.725,E2 -15951.725} C_VEL
LIN {X 0,Y 317.252,Z 559.769,A -85,B 0,C 180,E1 -15953.327,E2 -15953.327} C_VEL
LIN {X 0,Y 317.3,Z 550.008,A -85,B 0,C 180,E1 -15954.752,E2 -15954.752} C_VEL
LIN {X 0,Y 316.385,Z 540.688,A -85,B 0,C 180,E1 -15956.159,E2 -15956.159} C_VEL
LIN {X 0,Y 314.428,Z 530.222,A -85,B 0,C 180,E1 -15957.796,E2 -15957.796} C_VEL
LIN {X 0,Y 311.67,Z 520.178,A -85,B 0,C 180,E1 -15959.512,E2 -15959.512} C_VEL
LIN {X 0,Y 309.508,Z 513.567,A -85,B 0,C 180,E1 -15960.74,E2 -15960.74} C_VEL
LIN {X 0,Y 308.061,Z 510.323,A -85,B 0,C 180,E1 -15961.48,E2 -15961.48} C_VEL
LIN {X 0,Y 307.612,Z 507.934,A -85,B 0,C 180,E1 -15961.864,E2 -15961.864} C_VEL
LIN {X 0,Y 308.548,Z 504.271,A -85,B 0,C 180,E1 -15964.916,E2 -15964.916} C_VEL
LIN {X 0,Y 309.079,Z 501.227,A -85,B 0,C 180,E1 -15967.875,E2 -15967.875} C_VEL
LIN {X 0,Y 309.13,Z 499.769,A -85,B 0,C 180,E1 -15969.537,E2 -15969.537} C_VEL
LIN {X 0,Y 308.799,Z 497.142,A -85,B 0,C 180,E1 -15973.257,E2 -15973.257} C_VEL
LIN {X 0,Y 308.46,Z 495.303,A -85,B 0,C 180,E1 -15976.88,E2 -15976.88} C_VEL
LIN {X 0,Y 308.104,Z 494.062,A -85,B 0,C 180,E1 -15980.856,E2 -15980.856} C_VEL
LIN {X 0,Y 307.879,Z 493.65,A -85,B 0,C 180,E1 -15983.594,E2 -15983.594} C_VEL
LIN {X 0,Y 307.441,Z 493.625,A -85,B 0,C 180,E1 -15986.727,E2 -15986.727} C_VEL
LIN {X 0,Y 307.223,Z 493.828,A -85,B 0,C 180,E1 -15988.22,E2 -15988.22} C_VEL
LIN {X 0,Y 308.295,Z 496.499,A -85,B 0,C 180,E1 -15988.879,E2 -15988.879} C_VEL
LIN {X 0,Y 309.799,Z 498.214,A -85,B 0,C 180,E1 -15989.549,E2 -15989.549} C_VEL
LIN {X 0,Y 310.902,Z 500.678,A -85,B 0,C 180,E1 -15990.178,E2 -15990.178} C_VEL
LIN {X 0,Y 312.357,Z 502.463,A -85,B 0,C 180,E1 -15990.782,E2 -15990.782} C_VEL
LIN {X 0,Y 317.563,Z 513.759,A -85,B 0,C 180,E1 -15993.462,E2 -15993.462} C_VEL
LIN {X 0,Y 320.649,Z 523.141,A -85,B 0,C 180,E1 -15995.39,E2 -15995.39} C_VEL
LIN {X 0,Y 321.884,Z 528.892,A -85,B 0,C 180,E1 -15996.496,E2 -15996.496} C_VEL
LIN {X 0,Y 321.823,Z 531.227,A -85,B 0,C 180,E1 -15996.854,E2 -15996.854} C_VEL
LIN {X 0,Y 319.084,Z 542.099,A -85,B 0,C 180,E1 -15998.351,E2 -15998.351} C_VEL
LIN {X 0,Y 316.166,Z 552.798,A -85,B 0,C 180,E1 -16000.185,E2 -16000.185} C_VEL
LIN {X 0,Y 313.5,Z 561.565,A -85,B 0,C 180,E1 -16002.047,E2 -16002.047} C_VEL
LIN {X 0,Y 311.316,Z 568.714,A -85,B 0,C 180,E1 -16003.946,E2 -16003.946} C_VEL
LIN {X 0,Y 309.173,Z 575.468,A -85,B 0,C 180,E1 -16006.191,E2 -16006.191} C_VEL
LIN {X 0,Y 307.573,Z 580.024,A -85,B 0,C 180,E1 -16008.133,E2 -16008.133} C_VEL
LIN {X 0,Y 306.138,Z 584.456,A -85,B 0,C 180,E1 -16010.753,E2 -16010.753} C_VEL
LIN {X 0,Y 305.395,Z 586.099,A -85,B 0,C 180,E1 -16012.064,E2 -16012.064} C_VEL
LIN {X 0,Y 304.903,Z 587.275,A -85,B 0,C 180,E1 -16013.382,E2 -16013.382} C_VEL
LIN {X 0,Y 304.746,Z 588.043,A -85,B 0,C 180,E1 -16014.707,E2 -16014.707} C_VEL
LIN {X 0,Y 304.504,Z 588.447,A -85,B 0,C 180,E1 -16016.03,E2 -16016.03} C_VEL
LIN {X 0,Y 304.217,Z 588.464,A -85,B 0,C 180,E1 -16017.352,E2 -16017.352} C_VEL
LIN {X 0,Y 304.023,Z 588.047,A -85,B 0,C 180,E1 -16018.676,E2 -16018.676} C_VEL
LIN {X 0,Y 303.906,Z 587.237,A -85,B 0,C 180,E1 -16020,E2 -16020} C_VEL
LIN {X 0,Y 303.854,Z 586.033,A -85,B 0,C 180,E1 -16021.326,E2 -16021.326} C_VEL
LIN {X 0,Y 303.916,Z 583.405,A -85,B 0,C 180,E1 -16023.315,E2 -16023.315} C_VEL
LIN {X 0,Y 304.099,Z 579.777,A -85,B 0,C 180,E1 -16025.305,E2 -16025.305} C_VEL
LIN {X 0,Y 304.423,Z 574.819,A -85,B 0,C 180,E1 -16027.381,E2 -16027.381} C_VEL
LIN {X 0,Y 304.899,Z 567.971,A -85,B 0,C 180,E1 -16029.62,E2 -16029.62} C_VEL
LIN {X 0,Y 305.595,Z 560.359,A -85,B 0,C 180,E1 -16031.609,E2 -16031.609} C_VEL
LIN {X 0,Y 306.52,Z 550.939,A -85,B 0,C 180,E1 -16033.593,E2 -16033.593} C_VEL
LIN {X 0,Y 307.553,Z 540.274,A -85,B 0,C 180,E1 -16035.406,E2 -16035.406} C_VEL
LIN {X 0,Y 308.456,Z 530.878,A -85,B 0,C 180,E1 -16036.72,E2 -16036.72} C_VEL
LIN {X 0,Y 309.434,Z 519.519,A -85,B 0,C 180,E1 -16038.027,E2 -16038.027} C_VEL
LIN {X 0,Y 309.846,Z 513.018,A -85,B 0,C 180,E1 -16038.659,E2 -16038.659} C_VEL
LIN {X 0,Y 307.771,Z 501.824,A -85,B 0,C 180,E1 -16039.674,E2 -16039.674} C_VEL
LIN {X 0,Y 305.116,Z 488.134,A -85,B 0,C 180,E1 -16040.658,E2 -16040.658} C_VEL
LIN {X 0,Y 304.143,Z 482.976,A -85,B 0,C 180,E1 -16040.988,E2 -16040.988} C_VEL
LIN {X 0,Y 304.315,Z 478.681,A -85,B 0,C 180,E1 -16045.751,E2 -16045.751} C_VEL
LIN {X 0,Y 304.663,Z 478.533,A -85,B 0,C 180,E1 -16048.976,E2 -16048.976} C_VEL
LIN {X 0,Y 304.969,Z 478.496,A -85,B 0,C 180,E1 -16052.008,E2 -16052.008} C_VEL
LIN {X 0,Y 305.275,Z 478.456,A -85,B 0,C 180,E1 -16055.139,E2 -16055.139} C_VEL
LIN {X 0,Y 305.427,Z 478.44,A -85,B 0,C 180,E1 -16058.523,E2 -16058.523} C_VEL
LIN {X 0,Y 305.444,Z 478.436,A -85,B 0,C 180,E1 -16061.857,E2 -16061.857} C_VEL
LIN {X 0,Y 305.404,Z 478.44,A -85,B 0,C 180,E1 -16065.511,E2 -16065.511} C_VEL
LIN {X 0,Y 305.444,Z 478.439,A -85,B 0,C 180,E1 -16068.143,E2 -16068.143} C_VEL
LIN {X 0,Y 305.499,Z 478.428,A -85,B 0,C 180,E1 -16071.601,E2 -16071.601} C_VEL
LIN {X 0,Y 305.467,Z 478.432,A -85,B 0,C 180,E1 -16074.887,E2 -16074.887} C_VEL
LIN {X 0,Y 305.457,Z 478.436,A -85,B 0,C 180,E1 -16078.355,E2 -16078.355} C_VEL
LIN {X 0,Y 305.524,Z 478.424,A -85,B 0,C 180,E1 -16081.114,E2 -16081.114} C_VEL
LIN {X 0,Y 305.576,Z 478.423,A -85,B 0,C 180,E1 -16084.088,E2 -16084.088} C_VEL
LIN {X 0,Y 305.505,Z 478.429,A -85,B 0,C 180,E1 -16088.403,E2 -16088.403} C_VEL
LIN {X 0,Y 305.595,Z 478.416,A -85,B 0,C 180,E1 -16091.218,E2 -16091.218} C_VEL
LIN {X 0,Y 305.653,Z 478.409,A -85,B 0,C 180,E1 -16095.349,E2 -16095.349} C_VEL
LIN {X 0,Y 305.643,Z 478.41,A -85,B 0,C 180,E1 -16099.4,E2 -16099.4} C_VEL
LIN {X 0,Y 305.818,Z 478.393,A -85,B 0,C 180,E1 -16102.074,E2 -16102.074} C_VEL
LIN {X 0,Y 305.694,Z 478.403,A -85,B 0,C 180,E1 -16104.724,E2 -16104.724} C_VEL
LIN {X 0,Y 305.96,Z 478.371,A -85,B 0,C 180,E1 -16108.684,E2 -16108.684} C_VEL
LIN {X 0,Y 305.96,Z 478.371,A -85,B 0,C 180,E1 -16111.316,E2 -16111.316} C_VEL
LIN {X 0,Y 305.679,Z 478.405,A -85,B 0,C 180,E1 -16115.277,E2 -16115.277} C_VEL
LIN {X 0,Y 305.769,Z 478.399,A -85,B 0,C 180,E1 -16117.927,E2 -16117.927} C_VEL
LIN {X 0,Y 305.608,Z 478.419,A -85,B 0,C 180,E1 -16121.945,E2 -16121.945} C_VEL
LIN {X 0,Y 305.642,Z 478.41,A -85,B 0,C 180,E1 -16125.035,E2 -16125.035} C_VEL
LIN {X 0,Y 305.58,Z 478.419,A -85,B 0,C 180,E1 -16129.444,E2 -16129.444} C_VEL
LIN {X 0,Y 305.49,Z 478.428,A -85,B 0,C 180,E1 -16133.039,E2 -16133.039} C_VEL
LIN {X 0,Y 305.535,Z 478.425,A -85,B 0,C 180,E1 -16136.221,E2 -16136.221} C_VEL
LIN {X 0,Y 305.492,Z 478.429,A -85,B 0,C 180,E1 -16139.047,E2 -16139.047} C_VEL
LIN {X 0,Y 305.447,Z 478.438,A -85,B 0,C 180,E1 -16141.952,E2 -16141.952} C_VEL
LIN {X 0,Y 305.467,Z 478.432,A -85,B 0,C 180,E1 -16145.113,E2 -16145.113} C_VEL
LIN {X 0,Y 305.471,Z 478.431,A -85,B 0,C 180,E1 -16148.533,E2 -16148.533} C_VEL
LIN {X 0,Y 305.459,Z 478.433,A -85,B 0,C 180,E1 -16152.586,E2 -16152.586} C_VEL
LIN {X 0,Y 305.429,Z 478.437,A -85,B 0,C 180,E1 -16156.345,E2 -16156.345} C_VEL
LIN {X 0,Y 305.461,Z 478.436,A -85,B 0,C 180,E1 -16159.892,E2 -16159.892} C_VEL
LIN {X 0,Y 305.426,Z 478.442,A -85,B 0,C 180,E1 -16163.646,E2 -16163.646} C_VEL
LIN {X 0,Y 305.242,Z 478.459,A -85,B 0,C 180,E1 -16166.455,E2 -16166.455} C_VEL
LIN {X 0,Y 304.912,Z 478.505,A -85,B 0,C 180,E1 -16169.53,E2 -16169.53} C_VEL
LIN {X 0,Y 304.533,Z 478.548,A -85,B 0,C 180,E1 -16172.512,E2 -16172.512} C_VEL
LIN {X 0,Y 304.114,Z 478.673,A -85,B 0,C 180,E1 -16175.782,E2 -16175.782} C_VEL
LIN {X 0,Y 304.1,Z 482.216,A -85,B 0,C 180,E1 -16179.186,E2 -16179.186} C_VEL
LIN {X 0,Y 306.846,Z 496.946,A -85,B 0,C 180,E1 -16180.135,E2 -16180.135} C_VEL
LIN {X 0,Y 309.526,Z 510.966,A -85,B 0,C 180,E1 -16181.336,E2 -16181.336} C_VEL
LIN {X 0,Y 309.717,Z 514.241,A -85,B 0,C 180,E1 -16181.648,E2 -16181.648} C_VEL
LIN {X 0,Y 308.708,Z 527.189,A -85,B 0,C 180,E1 -16183.022,E2 -16183.022} C_VEL
LIN {X 0,Y 307.714,Z 537.796,A -85,B 0,C 180,E1 -16184.433,E2 -16184.433} C_VEL
LIN {X 0,Y 306.721,Z 547.985,A -85,B 0,C 180,E1 -16186.078,E2 -16186.078} C_VEL
LIN {X 0,Y 305.757,Z 557.845,A -85,B 0,C 180,E1 -16188.046,E2 -16188.046} C_VEL
LIN {X 0,Y 304.778,Z 561.535,A -85,B 0,C 180,E1 -16188.892,E2 -16188.892} C_VEL
LIN {X 0,Y 301.41,Z 567.064,A -85,B 0,C 180,E1 -16190.313,E2 -16190.313} C_VEL
LIN {X 0,Y 298.102,Z 572.022,A -85,B 0,C 180,E1 -16191.838,E2 -16191.838} C_VEL
LIN {X 0,Y 297.237,Z 574.789,A -85,B 0,C 180,E1 -16192.833,E2 -16192.833} C_VEL
LIN {X 0,Y 296.99,Z 578.969,A -85,B 0,C 180,E1 -16194.568,E2 -16194.568} C_VEL
LIN {X 0,Y 296.839,Z 582.821,A -85,B 0,C 180,E1 -16196.606,E2 -16196.606} C_VEL
LIN {X 0,Y 296.727,Z 585.629,A -85,B 0,C 180,E1 -16198.642,E2 -16198.642} C_VEL
LIN {X 0,Y 296.768,Z 586.987,A -85,B 0,C 180,E1 -16200,E2 -16200} C_VEL
LIN {X 0,Y 297.122,Z 588.404,A -85,B 0,C 180,E1 -16202.711,E2 -16202.711} C_VEL
LIN {X 0,Y 297.36,Z 588.535,A -85,B 0,C 180,E1 -16204.066,E2 -16204.066} C_VEL
LIN {X 0,Y 297.56,Z 588.261,A -85,B 0,C 180,E1 -16205.421,E2 -16205.421} C_VEL
LIN {X 0,Y 297.814,Z 587.573,A -85,B 0,C 180,E1 -16206.776,E2 -16206.776} C_VEL
LIN {X 0,Y 299.142,Z 585.025,A -85,B 0,C 180,E1 -16209.465,E2 -16209.465} C_VEL
LIN {X 0,Y 300.22,Z 582.032,A -85,B 0,C 180,E1 -16211.477,E2 -16211.477} C_VEL
LIN {X 0,Y 301.745,Z 578.016,A -85,B 0,C 180,E1 -16213.468,E2 -16213.468} C_VEL
LIN {X 0,Y 303.501,Z 572.993,A -85,B 0,C 180,E1 -16215.444,E2 -16215.444} C_VEL
LIN {X 0,Y 305.986,Z 565.553,A -85,B 0,C 180,E1 -16217.718,E2 -16217.718} C_VEL
LIN {X 0,Y 308.582,Z 557.706,A -85,B 0,C 180,E1 -16219.629,E2 -16219.629} C_VEL
LIN {X 0,Y 311.561,Z 548.1,A -85,B 0,C 180,E1 -16221.503,E2 -16221.503} C_VEL
LIN {X 0,Y 314.292,Z 538.077,A -85,B 0,C 180,E1 -16223.103,E2 -16223.103} C_VEL
LIN {X 0,Y 316.02,Z 531.664,A -85,B 0,C 180,E1 -16223.96,E2 -16223.96} C_VEL
LIN {X 0,Y 315.519,Z 526.949,A -85,B 0,C 180,E1 -16224.846,E2 -16224.846} C_VEL
LIN {X 0,Y 313.348,Z 518.188,A -85,B 0,C 180,E1 -16226.652,E2 -16226.652} C_VEL
LIN {X 0,Y 310.615,Z 510.707,A -85,B 0,C 180,E1 -16228.369,E2 -16228.369} C_VEL
LIN {X 0,Y 307.98,Z 504.784,A -85,B 0,C 180,E1 -16229.871,E2 -16229.871} C_VEL
LIN {X 0,Y 306.041,Z 500.968,A -85,B 0,C 180,E1 -16230.966,E2 -16230.966} C_VEL
LIN {X 0,Y 304.393,Z 498.219,A -85,B 0,C 180,E1 -16231.881,E2 -16231.881} C_VEL
LIN {X 0,Y 304.04,Z 497.342,A -85,B 0,C 180,E1 -16232.117,E2 -16232.117} C_VEL
LIN {X 0,Y 301.282,Z 493.442,A -85,B 0,C 180,E1 -16233.691,E2 -16233.691} C_VEL
LIN {X 0,Y 300.829,Z 492.099,A -85,B 0,C 180,E1 -16234.103,E2 -16234.103} C_VEL
LIN {X 0,Y 301.052,Z 490.973,A -85,B 0,C 180,E1 -16237.465,E2 -16237.465} C_VEL
LIN {X 0,Y 301.1,Z 490.486,A -85,B 0,C 180,E1 -16240.81,E2 -16240.81} C_VEL
LIN {X 0,Y 301.248,Z 490.617,A -85,B 0,C 180,E1 -16243.679,E2 -16243.679} C_VEL
LIN {X 0,Y 301.368,Z 491.316,A -85,B 0,C 180,E1 -16246.297,E2 -16246.297} C_VEL
LIN {X 0,Y 301.512,Z 492.91,A -85,B 0,C 180,E1 -16249.258,E2 -16249.258} C_VEL
LIN {X 0,Y 301.762,Z 495.638,A -85,B 0,C 180,E1 -16252.359,E2 -16252.359} C_VEL
LIN {X 0,Y 301.436,Z 498.873,A -85,B 0,C 180,E1 -16254.689,E2 -16254.689} C_VEL
LIN {X 0,Y 301.235,Z 501.315,A -85,B 0,C 180,E1 -16255.982,E2 -16255.982} C_VEL
LIN {X 0,Y 304.177,Z 509.214,A -85,B 0,C 180,E1 -16257.899,E2 -16257.899} C_VEL
LIN {X 0,Y 305.273,Z 512.795,A -85,B 0,C 180,E1 -16258.61,E2 -16258.61} C_VEL
LIN {X 0,Y 306.837,Z 518.979,A -85,B 0,C 180,E1 -16259.741,E2 -16259.741} C_VEL
LIN {X 0,Y 308.856,Z 529.23,A -85,B 0,C 180,E1 -16261.455,E2 -16261.455} C_VEL
LIN {X 0,Y 310.327,Z 540.855,A -85,B 0,C 180,E1 -16263.27,E2 -16263.27} C_VEL
LIN {X 0,Y 310.818,Z 553.473,A -85,B 0,C 180,E1 -16265.208,E2 -16265.208} C_VEL
LIN {X 0,Y 310.121,Z 562.82,A -85,B 0,C 180,E1 -16266.635,E2 -16266.635} C_VEL
LIN {X 0,Y 308.848,Z 570.936,A -85,B 0,C 180,E1 -16267.947,E2 -16267.947} C_VEL
LIN {X 0,Y 305.823,Z 581.757,A -85,B 0,C 180,E1 -16269.836,E2 -16269.836} C_VEL
LIN {X 0,Y 303.257,Z 590.932,A -85,B 0,C 180,E1 -16271.838,E2 -16271.838} C_VEL
LIN {X 0,Y 301.505,Z 597.008,A -85,B 0,C 180,E1 -16273.409,E2 -16273.409} C_VEL
LIN {X 0,Y 299.593,Z 604.284,A -85,B 0,C 180,E1 -16275.74,E2 -16275.74} C_VEL
LIN {X 0,Y 298.222,Z 609.349,A -85,B 0,C 180,E1 -16277.755,E2 -16277.755} C_VEL
LIN {X 0,Y 297.406,Z 613.349,A -85,B 0,C 180,E1 -16279.791,E2 -16279.791} C_VEL
LIN {X 0,Y 296.912,Z 616.38,A -85,B 0,C 180,E1 -16281.835,E2 -16281.835} C_VEL
LIN {X 0,Y 296.688,Z 619.004,A -85,B 0,C 180,E1 -16284.563,E2 -16284.563} C_VEL
LIN {X 0,Y 296.692,Z 619.682,A -85,B 0,C 180,E1 -16285.925,E2 -16285.925} C_VEL
LIN {X 0,Y 296.991,Z 619.807,A -85,B 0,C 180,E1 -16288.644,E2 -16288.644} C_VEL
LIN {X 0,Y 296.994,Z 620.81,A -85,B 0,C 180,E1 -16290,E2 -16290} C_VEL
LIN {X 0,Y 296.862,Z 621.357,A -85,B 0,C 180,E1 -16291.357,E2 -16291.357} C_VEL
LIN {X 0,Y 296.64,Z 621.229,A -85,B 0,C 180,E1 -16294.076,E2 -16294.076} C_VEL
LIN {X 0,Y 296.595,Z 620.43,A -85,B 0,C 180,E1 -16295.607,E2 -16295.607} C_VEL
LIN {X 0,Y 296.89,Z 617.954,A -85,B 0,C 180,E1 -16298.166,E2 -16298.166} C_VEL
LIN {X 0,Y 297.682,Z 613.765,A -85,B 0,C 180,E1 -16300.887,E2 -16300.887} C_VEL
LIN {X 0,Y 298.649,Z 609.478,A -85,B 0,C 180,E1 -16302.918,E2 -16302.918} C_VEL
LIN {X 0,Y 300.437,Z 603.095,A -85,B 0,C 180,E1 -16305.258,E2 -16305.258} C_VEL
LIN {X 0,Y 302.413,Z 595.237,A -85,B 0,C 180,E1 -16307.585,E2 -16307.585} C_VEL
LIN {X 0,Y 304.917,Z 586.968,A -85,B 0,C 180,E1 -16309.525,E2 -16309.525} C_VEL
LIN {X 0,Y 307.839,Z 577.046,A -85,B 0,C 180,E1 -16311.425,E2 -16311.425} C_VEL
LIN {X 0,Y 310.104,Z 568.366,A -85,B 0,C 180,E1 -16312.837,E2 -16312.837} C_VEL
LIN {X 0,Y 311.298,Z 559.089,A -85,B 0,C 180,E1 -16314.278,E2 -16314.278} C_VEL
LIN {X 0,Y 311.374,Z 550.478,A -85,B 0,C 180,E1 -16315.638,E2 -16315.638} C_VEL
LIN {X 0,Y 310.197,Z 539.032,A -85,B 0,C 180,E1 -16317.493,E2 -16317.493} C_VEL
LIN {X 0,Y 307.84,Z 527.669,A -85,B 0,C 180,E1 -16319.496,E2 -16319.496} C_VEL
LIN {X 0,Y 305.431,Z 518.994,A -85,B 0,C 180,E1 -16321.193,E2 -16321.193} C_VEL
LIN {X 0,Y 303.142,Z 512.403,A -85,B 0,C 180,E1 -16322.676,E2 -16322.676} C_VEL
LIN {X 0,Y 301.622,Z 508.714,A -85,B 0,C 180,E1 -16323.642,E2 -16323.642} C_VEL
LIN {X 0,Y 301.271,Z 506.687,A -85,B 0,C 180,E1 -16324.047,E2 -16324.047} C_VEL
LIN {X 0,Y 302.093,Z 503.342,A -85,B 0,C 180,E1 -16327.22,E2 -16327.22} C_VEL
LIN {X 0,Y 302.148,Z 501.053,A -85,B 0,C 180,E1 -16329.863,E2 -16329.863} C_VEL
LIN {X 0,Y 301.801,Z 498.422,A -85,B 0,C 180,E1 -16333.789,E2 -16333.789} C_VEL
LIN {X 0,Y 301.459,Z 496.684,A -85,B 0,C 180,E1 -16337.462,E2 -16337.462} C_VEL
LIN {X 0,Y 301.193,Z 495.639,A -85,B 0,C 180,E1 -16340.949,E2 -16340.949} C_VEL
LIN {X 0,Y 300.839,Z 495.191,A -85,B 0,C 180,E1 -16344.265,E2 -16344.265} C_VEL
LIN {X 0,Y 300.63,Z 495.277,A -85,B 0,C 180,E1 -16345.923,E2 -16345.923} C_VEL
LIN {X 0,Y 301.105,Z 496.737,A -85,B 0,C 180,E1 -16346.358,E2 -16346.358} C_VEL
LIN {X 0,Y 301.951,Z 498.178,A -85,B 0,C 180,E1 -16346.92,E2 -16346.92} C_VEL
LIN {X 0,Y 303.758,Z 499.966,A -85,B 0,C 180,E1 -16347.85,E2 -16347.85} C_VEL
LIN {X 0,Y 304.764,Z 502.42,A -85,B 0,C 180,E1 -16348.566,E2 -16348.566} C_VEL
LIN {X 0,Y 306.415,Z 504.691,A -85,B 0,C 180,E1 -16349.405,E2 -16349.405} C_VEL
LIN {X 0,Y 306.907,Z 506.072,A -85,B 0,C 180,E1 -16349.749,E2 -16349.749} C_VEL
LIN {X 0,Y 308.353,Z 508.317,A -85,B 0,C 180,E1 -16350.508,E2 -16350.508} C_VEL
LIN {X 0,Y 312.484,Z 517.889,A -85,B 0,C 180,E1 -16352.945,E2 -16352.945} C_VEL
LIN {X 0,Y 315.183,Z 526.863,A -85,B 0,C 180,E1 -16354.934,E2 -16354.934} C_VEL
LIN {X 0,Y 316.193,Z 532.605,A -85,B 0,C 180,E1 -16356.096,E2 -16356.096} C_VEL
LIN {X 0,Y 312.877,Z 544.968,A -85,B 0,C 180,E1 -16357.899,E2 -16357.899} C_VEL
LIN {X 0,Y 309.792,Z 555.152,A -85,B 0,C 180,E1 -16359.76,E2 -16359.76} C_VEL
LIN {X 0,Y 307,Z 563.526,A -85,B 0,C 180,E1 -16361.653,E2 -16361.653} C_VEL
LIN {X 0,Y 304.707,Z 570.437,A -85,B 0,C 180,E1 -16363.588,E2 -16363.588} C_VEL
LIN {X 0,Y 302.419,Z 576.842,A -85,B 0,C 180,E1 -16365.877,E2 -16365.877} C_VEL
LIN {X 0,Y 300.728,Z 581.193,A -85,B 0,C 180,E1 -16367.859,E2 -16367.859} C_VEL
LIN {X 0,Y 299.961,Z 583.522,A -85,B 0,C 180,E1 -16369.197,E2 -16369.197} C_VEL
LIN {X 0,Y 299.12,Z 585.612,A -85,B 0,C 180,E1 -16370.687,E2 -16370.687} C_VEL
LIN {X 0,Y 297.885,Z 588.001,A -85,B 0,C 180,E1 -16373.226,E2 -16373.226} C_VEL
LIN {X 0,Y 297.689,Z 588.691,A -85,B 0,C 180,E1 -16374.582,E2 -16374.582} C_VEL
LIN {X 0,Y 297.438,Z 589,A -85,B 0,C 180,E1 -16375.935,E2 -16375.935} C_VEL
LIN {X 0,Y 296.934,Z 588.398,A -85,B 0,C 180,E1 -16378.644,E2 -16378.644} C_VEL
LIN {X 0,Y 296.812,Z 587.512,A -85,B 0,C 180,E1 -16380,E2 -16380} C_VEL
LIN {X 0,Y 296.762,Z 586.21,A -85,B 0,C 180,E1 -16381.357,E2 -16381.357} C_VEL
LIN {X 0,Y 296.845,Z 583.461,A -85,B 0,C 180,E1 -16383.394,E2 -16383.394} C_VEL
LIN {X 0,Y 297.011,Z 579.68,A -85,B 0,C 180,E1 -16385.432,E2 -16385.432} C_VEL
LIN {X 0,Y 297.345,Z 574.78,A -85,B 0,C 180,E1 -16387.47,E2 -16387.47} C_VEL
LIN {X 0,Y 297.88,Z 567.471,A -85,B 0,C 180,E1 -16389.849,E2 -16389.849} C_VEL
LIN {X 0,Y 298.614,Z 559.653,A -85,B 0,C 180,E1 -16391.885,E2 -16391.885} C_VEL
LIN {X 0,Y 299.575,Z 549.967,A -85,B 0,C 180,E1 -16393.914,E2 -16393.914} C_VEL
LIN {X 0,Y 300.543,Z 540.157,A -85,B 0,C 180,E1 -16395.6,E2 -16395.6} C_VEL
LIN {X 0,Y 301.435,Z 530.907,A -85,B 0,C 180,E1 -16396.92,E2 -16396.92} C_VEL
LIN {X 0,Y 302.481,Z 519.263,A -85,B 0,C 180,E1 -16398.281,E2 -16398.281} C_VEL
LIN {X 0,Y 302.838,Z 514.221,A -85,B 0,C 180,E1 -16398.784,E2 -16398.784} C_VEL
LIN {X 0,Y 300.737,Z 502.561,A -85,B 0,C 180,E1 -16399.877,E2 -16399.877} C_VEL
LIN {X 0,Y 298.119,Z 489.053,A -85,B 0,C 180,E1 -16400.877,E2 -16400.877} C_VEL
LIN {X 0,Y 297.076,Z 483.361,A -85,B 0,C 180,E1 -16401.239,E2 -16401.239} C_VEL
LIN {X 0,Y 297.195,Z 479.837,A -85,B 0,C 180,E1 -16405.193,E2 -16405.193} C_VEL
LIN {X 0,Y 297.331,Z 479.451,A -85,B 0,C 180,E1 -16406.687,E2 -16406.687} C_VEL
LIN {X 0,Y 297.685,Z 479.402,A -85,B 0,C 180,E1 -16409.722,E2 -16409.722} C_VEL
LIN {X 0,Y 297.986,Z 479.364,A -85,B 0,C 180,E1 -16412.852,E2 -16412.852} C_VEL
LIN {X 0,Y 298.372,Z 479.317,A -85,B 0,C 180,E1 -16416.788,E2 -16416.788} C_VEL
LIN {X 0,Y 298.398,Z 479.312,A -85,B 0,C 180,E1 -16419.489,E2 -16419.489} C_VEL
LIN {X 0,Y 298.402,Z 479.312,A -85,B 0,C 180,E1 -16423.104,E2 -16423.104} C_VEL
LIN {X 0,Y 298.406,Z 479.312,A -85,B 0,C 180,E1 -16426.921,E2 -16426.921} C_VEL
LIN {X 0,Y 298.419,Z 479.309,A -85,B 0,C 180,E1 -16431.004,E2 -16431.004} C_VEL
LIN {X 0,Y 298.436,Z 479.31,A -85,B 0,C 180,E1 -16433.933,E2 -16433.933} C_VEL
LIN {X 0,Y 298.4,Z 479.315,A -85,B 0,C 180,E1 -16437.983,E2 -16437.983} C_VEL
LIN {X 0,Y 298.467,Z 479.306,A -85,B 0,C 180,E1 -16441.905,E2 -16441.905} C_VEL
LIN {X 0,Y 298.49,Z 479.301,A -85,B 0,C 180,E1 -16444.924,E2 -16444.924} C_VEL
LIN {X 0,Y 298.455,Z 479.305,A -85,B 0,C 180,E1 -16449.316,E2 -16449.316} C_VEL
LIN {X 0,Y 298.542,Z 479.299,A -85,B 0,C 180,E1 -16452.18,E2 -16452.18} C_VEL
LIN {X 0,Y 298.598,Z 479.287,A -85,B 0,C 180,E1 -16454.995,E2 -16454.995} C_VEL
LIN {X 0,Y 298.598,Z 479.287,A -85,B 0,C 180,E1 -16459.147,E2 -16459.147} C_VEL
LIN {X 0,Y 298.764,Z 479.271,A -85,B 0,C 180,E1 -16461.886,E2 -16461.886} C_VEL
LIN {X 0,Y 298.665,Z 479.279,A -85,B 0,C 180,E1 -16464.599,E2 -16464.599} C_VEL
LIN {X 0,Y 298.927,Z 479.247,A -85,B 0,C 180,E1 -16468.653,E2 -16468.653} C_VEL
LIN {X 0,Y 298.927,Z 479.247,A -85,B 0,C 180,E1 -16471.347,E2 -16471.347} C_VEL
LIN {X 0,Y 298.648,Z 479.281,A -85,B 0,C 180,E1 -16475.401,E2 -16475.401} C_VEL
LIN {X 0,Y 298.717,Z 479.276,A -85,B 0,C 180,E1 -16478.115,E2 -16478.115} C_VEL
LIN {X 0,Y 298.558,Z 479.294,A -85,B 0,C 180,E1 -16482.231,E2 -16482.231} C_VEL
LIN {X 0,Y 298.61,Z 479.286,A -85,B 0,C 180,E1 -16485.209,E2 -16485.209} C_VEL
LIN {X 0,Y 298.543,Z 479.295,A -85,B 0,C 180,E1 -16489.243,E2 -16489.243} C_VEL
LIN {X 0,Y 298.459,Z 479.307,A -85,B 0,C 180,E1 -16493.598,E2 -16493.598} C_VEL
LIN {X 0,Y 298.49,Z 479.301,A -85,B 0,C 180,E1 -16496.574,E2 -16496.574} C_VEL
LIN {X 0,Y 298.42,Z 479.313,A -85,B 0,C 180,E1 -16499.641,E2 -16499.641} C_VEL
LIN {X 0,Y 298.399,Z 479.312,A -85,B 0,C 180,E1 -16502.8,E2 -16502.8} C_VEL
LIN {X 0,Y 298.469,Z 479.303,A -85,B 0,C 180,E1 -16506.812,E2 -16506.812} C_VEL
LIN {X 0,Y 298.391,Z 479.313,A -85,B 0,C 180,E1 -16511.087,E2 -16511.087} C_VEL
LIN {X 0,Y 298.402,Z 479.312,A -85,B 0,C 180,E1 -16513.103,E2 -16513.103} C_VEL
LIN {X 0,Y 298.406,Z 479.311,A -85,B 0,C 180,E1 -16516.92,E2 -16516.92} C_VEL
LIN {X 0,Y 298.4,Z 479.312,A -85,B 0,C 180,E1 -16521.008,E2 -16521.008} C_VEL
LIN {X 0,Y 298.35,Z 479.321,A -85,B 0,C 180,E1 -16523.92,E2 -16523.92} C_VEL
LIN {X 0,Y 298.116,Z 479.348,A -85,B 0,C 180,E1 -16527.165,E2 -16527.165} C_VEL
LIN {X 0,Y 297.705,Z 479.399,A -85,B 0,C 180,E1 -16530.865,E2 -16530.865} C_VEL
LIN {X 0,Y 297.191,Z 479.462,A -85,B 0,C 180,E1 -16534.807,E2 -16534.807} C_VEL
LIN {X 0,Y 297.038,Z 479.637,A -85,B 0,C 180,E1 -16536.097,E2 -16536.097} C_VEL
LIN {X 0,Y 297.03,Z 482.576,A -85,B 0,C 180,E1 -16538.939,E2 -16538.939} C_VEL
LIN {X 0,Y 299.51,Z 496.176,A -85,B 0,C 180,E1 -16539.818,E2 -16539.818} C_VEL
LIN {X 0,Y 301.891,Z 508.769,A -85,B 0,C 180,E1 -16540.878,E2 -16540.878} C_VEL
LIN {X 0,Y 302.733,Z 513.918,A -85,B 0,C 180,E1 -16541.384,E2 -16541.384} C_VEL
LIN {X 0,Y 301.758,Z 526.435,A -85,B 0,C 180,E1 -16542.727,E2 -16542.727} C_VEL
LIN {X 0,Y 300.708,Z 537.639,A -85,B 0,C 180,E1 -16544.234,E2 -16544.234} C_VEL
LIN {X 0,Y 299.599,Z 548.805,A -85,B 0,C 180,E1 -16546.087,E2 -16546.087} C_VEL
LIN {X 0,Y 298.621,Z 558.604,A -85,B 0,C 180,E1 -16548.116,E2 -16548.116} C_VEL
LIN {X 0,Y 297.868,Z 566.605,A -85,B 0,C 180,E1 -16550.15,E2 -16550.15} C_VEL
LIN {X 0,Y 297.291,Z 573.987,A -85,B 0,C 180,E1 -16552.529,E2 -16552.529} C_VEL
LIN {X 0,Y 297.237,Z 574.789,A -85,B 0,C 180,E1 -16552.833,E2 -16552.833} C_VEL
LIN {X 0,Y 296.414,Z 577.384,A -85,B 0,C 180,E1 -16553.849,E2 -16553.849} C_VEL
LIN {X 0,Y 293.339,Z 580.998,A -85,B 0,C 180,E1 -16555.543,E2 -16555.543} C_VEL
LIN {X 0,Y 290.806,Z 583.466,A -85,B 0,C 180,E1 -16556.953,E2 -16556.953} C_VEL
LIN {X 0,Y 289.727,Z 585.071,A -85,B 0,C 180,E1 -16558.064,E2 -16558.064} C_VEL
LIN {X 0,Y 289.64,Z 585.506,A -85,B 0,C 180,E1 -16558.442,E2 -16558.442} C_VEL
LIN {X 0,Y 289.675,Z 587.176,A -85,B 0,C 180,E1 -16560,E2 -16560} C_VEL
LIN {X 0,Y 289.795,Z 588.22,A -85,B 0,C 180,E1 -16561.389,E2 -16561.389} C_VEL
LIN {X 0,Y 290.041,Z 588.814,A -85,B 0,C 180,E1 -16562.777,E2 -16562.777} C_VEL
LIN {X 0,Y 290.287,Z 589.023,A -85,B 0,C 180,E1 -16564.165,E2 -16564.165} C_VEL
LIN {X 0,Y 290.808,Z 588.311,A -85,B 0,C 180,E1 -16566.94,E2 -16566.94} C_VEL
LIN {X 0,Y 292.212,Z 585.924,A -85,B 0,C 180,E1 -16569.692,E2 -16569.692} C_VEL
LIN {X 0,Y 293.363,Z 583.118,A -85,B 0,C 180,E1 -16571.749,E2 -16571.749} C_VEL
LIN {X 0,Y 294.966,Z 579.338,A -85,B 0,C 180,E1 -16573.784,E2 -16573.784} C_VEL
LIN {X 0,Y 296.818,Z 574.507,A -85,B 0,C 180,E1 -16575.801,E2 -16575.801} C_VEL
LIN {X 0,Y 299.474,Z 567.45,A -85,B 0,C 180,E1 -16578.116,E2 -16578.116} C_VEL
LIN {X 0,Y 302.18,Z 559.916,A -85,B 0,C 180,E1 -16580.063,E2 -16580.063} C_VEL
LIN {X 0,Y 305.316,Z 550.766,A -85,B 0,C 180,E1 -16581.966,E2 -16581.966} C_VEL
LIN {X 0,Y 308.603,Z 539.875,A -85,B 0,C 180,E1 -16583.806,E2 -16583.806} C_VEL
LIN {X 0,Y 310.338,Z 533.72,A -85,B 0,C 180,E1 -16584.677,E2 -16584.677} C_VEL
LIN {X 0,Y 309.121,Z 525.723,A -85,B 0,C 180,E1 -16586.375,E2 -16586.375} C_VEL
LIN {X 0,Y 306.66,Z 517.212,A -85,B 0,C 180,E1 -16588.382,E2 -16588.382} C_VEL
LIN {X 0,Y 303.917,Z 510.274,A -85,B 0,C 180,E1 -16590.24,E2 -16590.24} C_VEL
LIN {X 0,Y 300.322,Z 502.93,A -85,B 0,C 180,E1 -16592.599,E2 -16592.599} C_VEL
LIN {X 0,Y 298.582,Z 500.382,A -85,B 0,C 180,E1 -16593.718,E2 -16593.718} C_VEL
LIN {X 0,Y 297.507,Z 498.182,A -85,B 0,C 180,E1 -16594.538,E2 -16594.538} C_VEL
LIN {X 0,Y 294.806,Z 494.783,A -85,B 0,C 180,E1 -16596.583,E2 -16596.583} C_VEL
LIN {X 0,Y 294.357,Z 493.543,A -85,B 0,C 180,E1 -16597.164,E2 -16597.164} C_VEL
LIN {X 0,Y 294.478,Z 493.161,A -85,B 0,C 180,E1 -16600.207,E2 -16600.207} C_VEL
LIN {X 0,Y 294.724,Z 493.433,A -85,B 0,C 180,E1 -16603.752,E2 -16603.752} C_VEL
LIN {X 0,Y 294.912,Z 494.226,A -85,B 0,C 180,E1 -16606.283,E2 -16606.283} C_VEL
LIN {X 0,Y 295.132,Z 496.249,A -85,B 0,C 180,E1 -16609.642,E2 -16609.642} C_VEL
LIN {X 0,Y 295.41,Z 499.2,A -85,B 0,C 180,E1 -16612.651,E2 -16612.651} C_VEL
LIN {X 0,Y 295.332,Z 500.066,A -85,B 0,C 180,E1 -16613.28,E2 -16613.28} C_VEL
LIN {X 0,Y 298.04,Z 507.703,A -85,B 0,C 180,E1 -16615.621,E2 -16615.621} C_VEL
LIN {X 0,Y 300.478,Z 514.914,A -85,B 0,C 180,E1 -16617.455,E2 -16617.455} C_VEL
LIN {X 0,Y 302.246,Z 522.879,A -85,B 0,C 180,E1 -16619.038,E2 -16619.038} C_VEL
LIN {X 0,Y 304.234,Z 536.063,A -85,B 0,C 180,E1 -16621.381,E2 -16621.381} C_VEL
LIN {X 0,Y 304.951,Z 547.661,A -85,B 0,C 180,E1 -16623.286,E2 -16623.286} C_VEL
LIN {X 0,Y 304.811,Z 557.816,A -85,B 0,C 180,E1 -16624.946,E2 -16624.946} C_VEL
LIN {X 0,Y 303.283,Z 569.054,A -85,B 0,C 180,E1 -16626.8,E2 -16626.8} C_VEL
LIN {X 0,Y 301.298,Z 576.462,A -85,B 0,C 180,E1 -16628.086,E2 -16628.086} C_VEL
LIN {X 0,Y 298.356,Z 586.134,A -85,B 0,C 180,E1 -16630.028,E2 -16630.028} C_VEL
LIN {X 0,Y 295.478,Z 595.177,A -85,B 0,C 180,E1 -16632.28,E2 -16632.28} C_VEL
LIN {X 0,Y 293.356,Z 602.886,A -85,B 0,C 180,E1 -16634.72,E2 -16634.72} C_VEL
LIN {X 0,Y 291.725,Z 608.086,A -85,B 0,C 180,E1 -16636.77,E2 -16636.77} C_VEL
LIN {X 0,Y 290.405,Z 613.405,A -85,B 0,C 180,E1 -16639.542,E2 -16639.542} C_VEL
LIN {X 0,Y 289.862,Z 616.271,A -85,B 0,C 180,E1 -16641.635,E2 -16641.635} C_VEL
LIN {X 0,Y 289.602,Z 618.594,A -85,B 0,C 180,E1 -16644.257,E2 -16644.257} C_VEL
LIN {X 0,Y 289.604,Z 619.269,A -85,B 0,C 180,E1 -16645.825,E2 -16645.825} C_VEL
LIN {X 0,Y 289.906,Z 619.248,A -85,B 0,C 180,E1 -16648.611,E2 -16648.611} C_VEL
LIN {X 0,Y 289.939,Z 620.147,A -85,B 0,C 180,E1 -16650,E2 -16650} C_VEL
LIN {X 0,Y 289.773,Z 620.789,A -85,B 0,C 180,E1 -16651.39,E2 -16651.39} C_VEL
LIN {X 0,Y 289.551,Z 620.802,A -85,B 0,C 180,E1 -16654.176,E2 -16654.176} C_VEL
LIN {X 0,Y 289.602,Z 619.229,A -85,B 0,C 180,E1 -16656.969,E2 -16656.969} C_VEL
LIN {X 0,Y 290.21,Z 616.026,A -85,B 0,C 180,E1 -16659.76,E2 -16659.76} C_VEL
LIN {X 0,Y 291.286,Z 611.201,A -85,B 0,C 180,E1 -16662.542,E2 -16662.542} C_VEL
LIN {X 0,Y 292.75,Z 606.429,A -85,B 0,C 180,E1 -16664.6,E2 -16664.6} C_VEL
LIN {X 0,Y 294.73,Z 599.497,A -85,B 0,C 180,E1 -16666.984,E2 -16666.984} C_VEL
LIN {X 0,Y 297.015,Z 592.228,A -85,B 0,C 180,E1 -16668.987,E2 -16668.987} C_VEL
LIN {X 0,Y 299.809,Z 583.592,A -85,B 0,C 180,E1 -16670.946,E2 -16670.946} C_VEL
LIN {X 0,Y 303.097,Z 573.163,A -85,B 0,C 180,E1 -16672.854,E2 -16672.854} C_VEL
LIN {X 0,Y 305.061,Z 563.347,A -85,B 0,C 180,E1 -16674.5,E2 -16674.5} C_VEL
LIN {X 0,Y 305.555,Z 554.85,A -85,B 0,C 180,E1 -16675.914,E2 -16675.914} C_VEL
LIN {X 0,Y 305.026,Z 544.842,A -85,B 0,C 180,E1 -16677.654,E2 -16677.654} C_VEL
LIN {X 0,Y 303.777,Z 535.866,A -85,B 0,C 180,E1 -16679.288,E2 -16679.288} C_VEL
LIN {X 0,Y 301.909,Z 527.33,A -85,B 0,C 180,E1 -16681.006,E2 -16681.006} C_VEL
LIN {X 0,Y 299.551,Z 518.594,A -85,B 0,C 180,E1 -16682.969,E2 -16682.969} C_VEL
LIN {X 0,Y 297.801,Z 513.563,A -85,B 0,C 180,E1 -16684.311,E2 -16684.311} C_VEL
LIN {X 0,Y 297.659,Z 512.61,A -85,B 0,C 180,E1 -16684.518,E2 -16684.518} C_VEL
LIN {X 0,Y 295.611,Z 508.108,A -85,B 0,C 180,E1 -16686.067,E2 -16686.067} C_VEL
LIN {X 0,Y 295.033,Z 505.141,A -85,B 0,C 180,E1 -16686.918,E2 -16686.918} C_VEL
LIN {X 0,Y 295.198,Z 503.926,A -85,B 0,C 180,E1 -16688.243,E2 -16688.243} C_VEL
LIN {X 0,Y 295.159,Z 502.235,A -85,B 0,C 180,E1 -16690.364,E2 -16690.364} C_VEL
LIN {X 0,Y 294.893,Z 500.054,A -85,B 0,C 180,E1 -16693.721,E2 -16693.721} C_VEL
LIN {X 0,Y 294.529,Z 498.2,A -85,B 0,C 180,E1 -16697.708,E2 -16697.708} C_VEL
LIN {X 0,Y 294.353,Z 497.513,A -85,B 0,C 180,E1 -16699.86,E2 -16699.86} C_VEL
LIN {X 0,Y 294.115,Z 497.015,A -85,B 0,C 180,E1 -16702.839,E2 -16702.839} C_VEL
LIN {X 0,Y 295.222,Z 499.51,A -85,B 0,C 180,E1 -16704.037,E2 -16704.037} C_VEL
LIN {X 0,Y 297.165,Z 501.336,A -85,B 0,C 180,E1 -16705.417,E2 -16705.417} C_VEL
LIN {X 0,Y 298.652,Z 504.23,A -85,B 0,C 180,E1 -16706.606,E2 -16706.606} C_VEL
LIN {X 0,Y 300.118,Z 505.817,A -85,B 0,C 180,E1 -16707.462,E2 -16707.462} C_VEL
LIN {X 0,Y 301.12,Z 508.24,A -85,B 0,C 180,E1 -16708.239,E2 -16708.239} C_VEL
LIN {X 0,Y 301.971,Z 509.365,A -85,B 0,C 180,E1 -16708.742,E2 -16708.742} C_VEL
LIN {X 0,Y 304.882,Z 515.521,A -85,B 0,C 180,E1 -16710.662,E2 -16710.662} C_VEL
LIN {X 0,Y 308.306,Z 524.86,A -85,B 0,C 180,E1 -16713.119,E2 -16713.119} C_VEL
LIN {X 0,Y 310.177,Z 532.971,A -85,B 0,C 180,E1 -16715.003,E2 -16715.003} C_VEL
LIN {X 0,Y 310.363,Z 534.298,A -85,B 0,C 180,E1 -16715.289,E2 -16715.289} C_VEL
LIN {X 0,Y 309.822,Z 537.449,A -85,B 0,C 180,E1 -16715.783,E2 -16715.783} C_VEL
LIN {X 0,Y 306.681,Z 547.833,A -85,B 0,C 180,E1 -16717.428,E2 -16717.428} C_VEL
LIN {X 0,Y 303.443,Z 557.551,A -85,B 0,C 180,E1 -16719.317,E2 -16719.317} C_VEL
LIN {X 0,Y 300.519,Z 565.563,A -85,B 0,C 180,E1 -16721.243,E2 -16721.243} C_VEL
LIN {X 0,Y 297.69,Z 573.08,A -85,B 0,C 180,E1 -16723.543,E2 -16723.543} C_VEL
LIN {X 0,Y 295.7,Z 578.283,A -85,B 0,C 180,E1 -16725.549,E2 -16725.549} C_VEL
LIN {X 0,Y 293.903,Z 582.416,A -85,B 0,C 180,E1 -16727.572,E2 -16727.572} C_VEL
LIN {X 0,Y 293.077,Z 584.589,A -85,B 0,C 180,E1 -16728.94,E2 -16728.94} C_VEL
LIN {X 0,Y 291.472,Z 587.758,A -85,B 0,C 180,E1 -16731.682,E2 -16731.682} C_VEL
LIN {X 0,Y 290.873,Z 588.76,A -85,B 0,C 180,E1 -16733.062,E2 -16733.062} C_VEL
LIN {X 0,Y 290.634,Z 589.327,A -85,B 0,C 180,E1 -16734.45,E2 -16734.45} C_VEL
LIN {X 0,Y 290.368,Z 589.505,A -85,B 0,C 180,E1 -16735.836,E2 -16735.836} C_VEL
LIN {X 0,Y 289.845,Z 588.74,A -85,B 0,C 180,E1 -16738.611,E2 -16738.611} C_VEL
LIN {X 0,Y 289.717,Z 587.746,A -85,B 0,C 180,E1 -16740,E2 -16740} C_VEL
LIN {X 0,Y 289.672,Z 586.323,A -85,B 0,C 180,E1 -16741.391,E2 -16741.391} C_VEL
LIN {X 0,Y 289.777,Z 583.417,A -85,B 0,C 180,E1 -16743.476,E2 -16743.476} C_VEL
LIN {X 0,Y 289.947,Z 578.621,A -85,B 0,C 180,E1 -16745.966,E2 -16745.966} C_VEL
LIN {X 0,Y 290.395,Z 572.51,A -85,B 0,C 180,E1 -16748.35,E2 -16748.35} C_VEL
LIN {X 0,Y 291.07,Z 564.428,A -85,B 0,C 180,E1 -16750.786,E2 -16750.786} C_VEL
LIN {X 0,Y 291.897,Z 555.777,A -85,B 0,C 180,E1 -16752.869,E2 -16752.869} C_VEL
LIN {X 0,Y 293.033,Z 545.097,A -85,B 0,C 180,E1 -16754.941,E2 -16754.941} C_VEL
LIN {X 0,Y 294.201,Z 534.097,A -85,B 0,C 180,E1 -16756.659,E2 -16756.659} C_VEL
LIN {X 0,Y 295.258,Z 521.873,A -85,B 0,C 180,E1 -16758.205,E2 -16758.205} C_VEL
LIN {X 0,Y 295.752,Z 515.363,A -85,B 0,C 180,E1 -16758.892,E2 -16758.892} C_VEL
LIN {X 0,Y 294.403,Z 506.887,A -85,B 0,C 180,E1 -16759.734,E2 -16759.734} C_VEL
LIN {X 0,Y 292.016,Z 494.407,A -85,B 0,C 180,E1 -16760.767,E2 -16760.767} C_VEL
LIN {X 0,Y 290.011,Z 483.742,A -85,B 0,C 180,E1 -16761.502,E2 -16761.502} C_VEL
LIN {X 0,Y 290.053,Z 481.255,A -85,B 0,C 180,E1 -16764.325,E2 -16764.325} C_VEL
LIN {X 0,Y 290.217,Z 480.336,A -85,B 0,C 180,E1 -16765.843,E2 -16765.843} C_VEL
LIN {X 0,Y 290.616,Z 480.282,A -85,B 0,C 180,E1 -16769.472,E2 -16769.472} C_VEL
LIN {X 0,Y 290.907,Z 480.25,A -85,B 0,C 180,E1 -16772.267,E2 -16772.267} C_VEL
LIN {X 0,Y 291.182,Z 480.211,A -85,B 0,C 180,E1 -16775.4,E2 -16775.4} C_VEL
LIN {X 0,Y 291.319,Z 480.194,A -85,B 0,C 180,E1 -16777.239,E2 -16777.239} C_VEL
